LIN {X 0,Y 361.859,Z 339.019,A -85,B 0,C 180,E1 -13169.074,E2 -13169.074} C_VEL
LIN {X 0,Y 361.85,Z 339.033,A -85,B 0,C 180,E1 -13172.945,E2 -13172.945} C_VEL
LIN {X 0,Y 361.866,Z 339.018,A -85,B 0,C 180,E1 -13175.637,E2 -13175.637} C_VEL
LIN {X 0,Y 361.827,Z 339.039,A -85,B 0,C 180,E1 -13179.018,E2 -13179.018} C_VEL
LIN {X 0,Y 361.832,Z 339.037,A -85,B 0,C 180,E1 -13182.83,E2 -13182.83} C_VEL
LIN {X 0,Y 361.815,Z 339.032,A -85,B 0,C 180,E1 -13185.948,E2 -13185.948} C_VEL
LIN {X 0,Y 361.813,Z 339.037,A -85,B 0,C 180,E1 -13189.25,E2 -13189.25} C_VEL
LIN {X 0,Y 361.863,Z 339.037,A -85,B 0,C 180,E1 -13192.981,E2 -13192.981} C_VEL
LIN {X 0,Y 361.888,Z 339.154,A -85,B 0,C 180,E1 -13194.653,E2 -13194.653} C_VEL
LIN {X 0,Y 364.151,Z 348.355,A -85,B 0,C 180,E1 -13197.305,E2 -13197.305} C_VEL
LIN {X 0,Y 374.278,Z 371.025,A -85,B 0,C 180,E1 -13198.692,E2 -13198.692} C_VEL
LIN {X 0,Y 376.076,Z 376.225,A -85,B 0,C 180,E1 -13198.951,E2 -13198.951} C_VEL
LIN {X 0,Y 376.861,Z 380.502,A -85,B 0,C 180,E1 -13199.105,E2 -13199.105} C_VEL
LIN {X 0,Y 374.503,Z 484.658,A -85,B 0,C 180,E1 -13201.142,E2 -13201.142} C_VEL
LIN {X 0,Y 373.689,Z 499.489,A -85,B 0,C 180,E1 -13201.648,E2 -13201.648} C_VEL
LIN {X 0,Y 372.585,Z 513.31,A -85,B 0,C 180,E1 -13202.343,E2 -13202.343} C_VEL
LIN {X 0,Y 371.503,Z 525.302,A -85,B 0,C 180,E1 -13203.149,E2 -13203.149} C_VEL
LIN {X 0,Y 370.031,Z 538.195,A -85,B 0,C 180,E1 -13204.249,E2 -13204.249} C_VEL
LIN {X 0,Y 368.437,Z 549.874,A -85,B 0,C 180,E1 -13205.488,E2 -13205.488} C_VEL
LIN {X 0,Y 367.047,Z 560.816,A -85,B 0,C 180,E1 -13206.927,E2 -13206.927} C_VEL
LIN {X 0,Y 365.472,Z 571.118,A -85,B 0,C 180,E1 -13208.57,E2 -13208.57} C_VEL
LIN {X 0,Y 364.126,Z 579.801,A -85,B 0,C 180,E1 -13210.259,E2 -13210.259} C_VEL
LIN {X 0,Y 362.938,Z 588.089,A -85,B 0,C 180,E1 -13212.243,E2 -13212.243} C_VEL
LIN {X 0,Y 361.932,Z 594.713,A -85,B 0,C 180,E1 -13214.225,E2 -13214.225} C_VEL
LIN {X 0,Y 361.377,Z 599.273,A -85,B 0,C 180,E1 -13215.93,E2 -13215.93} C_VEL
LIN {X 0,Y 360.876,Z 602.89,A -85,B 0,C 180,E1 -13217.63,E2 -13217.63} C_VEL
LIN {X 0,Y 360.463,Z 606.411,A -85,B 0,C 180,E1 -13219.894,E2 -13219.894} C_VEL
LIN {X 0,Y 360.324,Z 608.525,A -85,B 0,C 180,E1 -13222.153,E2 -13222.153} C_VEL
LIN {X 0,Y 360.339,Z 609.296,A -85,B 0,C 180,E1 -13224.404,E2 -13224.404} C_VEL
LIN {X 0,Y 360.306,Z 608.752,A -85,B 0,C 180,E1 -13226.645,E2 -13226.645} C_VEL
LIN {X 0,Y 360.396,Z 606.887,A -85,B 0,C 180,E1 -13228.883,E2 -13228.883} C_VEL
LIN {X 0,Y 360.58,Z 603.647,A -85,B 0,C 180,E1 -13231.117,E2 -13231.117} C_VEL
LIN {X 0,Y 360.995,Z 598.934,A -85,B 0,C 180,E1 -13233.348,E2 -13233.348} C_VEL
LIN {X 0,Y 361.574,Z 594.379,A -85,B 0,C 180,E1 -13235.018,E2 -13235.018} C_VEL
LIN {X 0,Y 362.267,Z 587.776,A -85,B 0,C 180,E1 -13236.964,E2 -13236.964} C_VEL
LIN {X 0,Y 363.207,Z 579.566,A -85,B 0,C 180,E1 -13238.905,E2 -13238.905} C_VEL
LIN {X 0,Y 363.908,Z 572.559,A -85,B 0,C 180,E1 -13240.291,E2 -13240.291} C_VEL
LIN {X 0,Y 365.328,Z 562.556,A -85,B 0,C 180,E1 -13241.935,E2 -13241.935} C_VEL
LIN {X 0,Y 366.604,Z 551.394,A -85,B 0,C 180,E1 -13243.441,E2 -13243.441} C_VEL
LIN {X 0,Y 367.903,Z 538.895,A -85,B 0,C 180,E1 -13244.803,E2 -13244.803} C_VEL
LIN {X 0,Y 369.111,Z 526.476,A -85,B 0,C 180,E1 -13245.885,E2 -13245.885} C_VEL
LIN {X 0,Y 369.72,Z 519.402,A -85,B 0,C 180,E1 -13246.397,E2 -13246.397} C_VEL
LIN {X 0,Y 369.535,Z 514.034,A -85,B 0,C 180,E1 -13246.781,E2 -13246.781} C_VEL
LIN {X 0,Y 367.497,Z 505.26,A -85,B 0,C 180,E1 -13247.428,E2 -13247.428} C_VEL
LIN {X 0,Y 365.305,Z 496.282,A -85,B 0,C 180,E1 -13247.988,E2 -13247.988} C_VEL
LIN {X 0,Y 364.865,Z 490.597,A -85,B 0,C 180,E1 -13248.231,E2 -13248.231} C_VEL
LIN {X 0,Y 365.345,Z 475.344,A -85,B 0,C 180,E1 -13248.615,E2 -13248.615} C_VEL
LIN {X 0,Y 367.351,Z 379.982,A -85,B 0,C 180,E1 -13250.471,E2 -13250.471} C_VEL
LIN {X 0,Y 365.287,Z 370.104,A -85,B 0,C 180,E1 -13250.822,E2 -13250.822} C_VEL
LIN {X 0,Y 356.698,Z 348.251,A -85,B 0,C 180,E1 -13251.941,E2 -13251.941} C_VEL
LIN {X 0,Y 354.827,Z 339.915,A -85,B 0,C 180,E1 -13254.262,E2 -13254.262} C_VEL
LIN {X 0,Y 354.796,Z 339.921,A -85,B 0,C 180,E1 -13257.104,E2 -13257.104} C_VEL
LIN {X 0,Y 354.796,Z 339.911,A -85,B 0,C 180,E1 -13259.684,E2 -13259.684} C_VEL
LIN {X 0,Y 354.81,Z 339.912,A -85,B 0,C 180,E1 -13263.702,E2 -13263.702} C_VEL
LIN {X 0,Y 354.794,Z 339.916,A -85,B 0,C 180,E1 -13266.46,E2 -13266.46} C_VEL
LIN {X 0,Y 354.771,Z 339.916,A -85,B 0,C 180,E1 -13269.412,E2 -13269.412} C_VEL
LIN {X 0,Y 354.784,Z 339.918,A -85,B 0,C 180,E1 -13272.866,E2 -13272.866} C_VEL
LIN {X 0,Y 354.765,Z 339.916,A -85,B 0,C 180,E1 -13276.103,E2 -13276.103} C_VEL
LIN {X 0,Y 354.765,Z 339.916,A -85,B 0,C 180,E1 -13279.175,E2 -13279.175} C_VEL
LIN {X 0,Y 354.801,Z 339.91,A -85,B 0,C 180,E1 -13282.404,E2 -13282.404} C_VEL
LIN {X 0,Y 354.813,Z 339.913,A -85,B 0,C 180,E1 -13284.94,E2 -13284.94} C_VEL
LIN {X 0,Y 354.796,Z 339.91,A -85,B 0,C 180,E1 -13288.405,E2 -13288.405} C_VEL
LIN {X 0,Y 354.791,Z 339.91,A -85,B 0,C 180,E1 -13291.613,E2 -13291.613} C_VEL
LIN {X 0,Y 354.807,Z 339.912,A -85,B 0,C 180,E1 -13295.419,E2 -13295.419} C_VEL
LIN {X 0,Y 354.824,Z 339.888,A -85,B 0,C 180,E1 -13299.113,E2 -13299.113} C_VEL
LIN {X 0,Y 354.854,Z 339.907,A -85,B 0,C 180,E1 -13302.717,E2 -13302.717} C_VEL
LIN {X 0,Y 354.943,Z 339.89,A -85,B 0,C 180,E1 -13306.254,E2 -13306.254} C_VEL
LIN {X 0,Y 354.959,Z 339.867,A -85,B 0,C 180,E1 -13309.735,E2 -13309.735} C_VEL
LIN {X 0,Y 355.091,Z 339.875,A -85,B 0,C 180,E1 -13313.18,E2 -13313.18} C_VEL
LIN {X 0,Y 355.237,Z 339.857,A -85,B 0,C 180,E1 -13317.732,E2 -13317.732} C_VEL
LIN {X 0,Y 355.175,Z 339.859,A -85,B 0,C 180,E1 -13321.133,E2 -13321.133} C_VEL
LIN {X 0,Y 355.231,Z 339.861,A -85,B 0,C 180,E1 -13322.267,E2 -13322.267} C_VEL
LIN {X 0,Y 355.092,Z 339.875,A -85,B 0,C 180,E1 -13326.82,E2 -13326.82} C_VEL
LIN {X 0,Y 354.959,Z 339.892,A -85,B 0,C 180,E1 -13330.264,E2 -13330.264} C_VEL
LIN {X 0,Y 354.945,Z 339.893,A -85,B 0,C 180,E1 -13334.019,E2 -13334.019} C_VEL
LIN {X 0,Y 354.925,Z 339.896,A -85,B 0,C 180,E1 -13338.108,E2 -13338.108} C_VEL
LIN {X 0,Y 354.835,Z 339.908,A -85,B 0,C 180,E1 -13342.106,E2 -13342.106} C_VEL
LIN {X 0,Y 354.872,Z 339.905,A -85,B 0,C 180,E1 -13345.829,E2 -13345.829} C_VEL
LIN {X 0,Y 354.809,Z 339.913,A -85,B 0,C 180,E1 -13349.682,E2 -13349.682} C_VEL
LIN {X 0,Y 354.832,Z 339.914,A -85,B 0,C 180,E1 -13353.682,E2 -13353.682} C_VEL
LIN {X 0,Y 354.803,Z 339.915,A -85,B 0,C 180,E1 -13356.459,E2 -13356.459} C_VEL
LIN {X 0,Y 354.825,Z 339.913,A -85,B 0,C 180,E1 -13359.423,E2 -13359.423} C_VEL
LIN {X 0,Y 354.789,Z 339.917,A -85,B 0,C 180,E1 -13362.867,E2 -13362.867} C_VEL
LIN {X 0,Y 354.768,Z 339.918,A -85,B 0,C 180,E1 -13366.103,E2 -13366.103} C_VEL
LIN {X 0,Y 354.789,Z 339.918,A -85,B 0,C 180,E1 -13369.179,E2 -13369.179} C_VEL
LIN {X 0,Y 354.809,Z 339.918,A -85,B 0,C 180,E1 -13372.402,E2 -13372.402} C_VEL
LIN {X 0,Y 354.813,Z 339.918,A -85,B 0,C 180,E1 -13374.941,E2 -13374.941} C_VEL
LIN {X 0,Y 354.832,Z 339.964,A -85,B 0,C 180,E1 -13377.039,E2 -13377.039} C_VEL
LIN {X 0,Y 357.952,Z 353.28,A -85,B 0,C 180,E1 -13380.365,E2 -13380.365} C_VEL
LIN {X 0,Y 360.186,Z 364.464,A -85,B 0,C 180,E1 -13383.021,E2 -13383.021} C_VEL
LIN {X 0,Y 360.211,Z 366.003,A -85,B 0,C 180,E1 -13383.361,E2 -13383.361} C_VEL
LIN {X 0,Y 365.124,Z 394.057,A -85,B 0,C 180,E1 -13384.311,E2 -13384.311} C_VEL
LIN {X 0,Y 366.939,Z 405.452,A -85,B 0,C 180,E1 -13384.672,E2 -13384.672} C_VEL
LIN {X 0,Y 364.837,Z 504.382,A -85,B 0,C 180,E1 -13386.628,E2 -13386.628} C_VEL
LIN {X 0,Y 364.064,Z 518.99,A -85,B 0,C 180,E1 -13387.139,E2 -13387.139} C_VEL
LIN {X 0,Y 363.033,Z 532.395,A -85,B 0,C 180,E1 -13387.821,E2 -13387.821} C_VEL
LIN {X 0,Y 361.759,Z 546.228,A -85,B 0,C 180,E1 -13388.772,E2 -13388.772} C_VEL
LIN {X 0,Y 360.495,Z 558.957,A -85,B 0,C 180,E1 -13389.903,E2 -13389.903} C_VEL
LIN {X 0,Y 359.032,Z 570.399,A -85,B 0,C 180,E1 -13391.156,E2 -13391.156} C_VEL
LIN {X 0,Y 357.718,Z 580.918,A -85,B 0,C 180,E1 -13392.566,E2 -13392.566} C_VEL
LIN {X 0,Y 356.386,Z 591.377,A -85,B 0,C 180,E1 -13394.267,E2 -13394.267} C_VEL
LIN {X 0,Y 355.49,Z 600.131,A -85,B 0,C 180,E1 -13396.011,E2 -13396.011} C_VEL
LIN {X 0,Y 354.542,Z 608.246,A -85,B 0,C 180,E1 -13397.987,E2 -13397.987} C_VEL
LIN {X 0,Y 353.928,Z 614.029,A -85,B 0,C 180,E1 -13399.705,E2 -13399.705} C_VEL
LIN {X 0,Y 353.584,Z 618.743,A -85,B 0,C 180,E1 -13401.427,E2 -13401.427} C_VEL
LIN {X 0,Y 353.4,Z 622.55,A -85,B 0,C 180,E1 -13403.147,E2 -13403.147} C_VEL
LIN {X 0,Y 353.269,Z 626.266,A -85,B 0,C 180,E1 -13405.436,E2 -13405.436} C_VEL
LIN {X 0,Y 353.181,Z 628.562,A -85,B 0,C 180,E1 -13407.719,E2 -13407.719} C_VEL
LIN {X 0,Y 353.261,Z 629.505,A -85,B 0,C 180,E1 -13410,E2 -13410} C_VEL
LIN {X 0,Y 353.168,Z 629.106,A -85,B 0,C 180,E1 -13412.281,E2 -13412.281} C_VEL
LIN {X 0,Y 353.247,Z 627.377,A -85,B 0,C 180,E1 -13414.565,E2 -13414.565} C_VEL
LIN {X 0,Y 353.402,Z 624.276,A -85,B 0,C 180,E1 -13416.853,E2 -13416.853} C_VEL
LIN {X 0,Y 353.737,Z 619.722,A -85,B 0,C 180,E1 -13419.146,E2 -13419.146} C_VEL
LIN {X 0,Y 354.188,Z 615.221,A -85,B 0,C 180,E1 -13420.866,E2 -13420.866} C_VEL
LIN {X 0,Y 355.165,Z 608.756,A -85,B 0,C 180,E1 -13422.863,E2 -13422.863} C_VEL
LIN {X 0,Y 356.139,Z 600.743,A -85,B 0,C 180,E1 -13424.865,E2 -13424.865} C_VEL
LIN {X 0,Y 357.459,Z 592.378,A -85,B 0,C 180,E1 -13426.564,E2 -13426.564} C_VEL
LIN {X 0,Y 359.051,Z 582.325,A -85,B 0,C 180,E1 -13428.251,E2 -13428.251} C_VEL
LIN {X 0,Y 360.848,Z 571.117,A -85,B 0,C 180,E1 -13429.78,E2 -13429.78} C_VEL
LIN {X 0,Y 362.413,Z 559.991,A -85,B 0,C 180,E1 -13431.024,E2 -13431.024} C_VEL
LIN {X 0,Y 363.899,Z 547.901,A -85,B 0,C 180,E1 -13432.123,E2 -13432.123} C_VEL
LIN {X 0,Y 365.294,Z 534.497,A -85,B 0,C 180,E1 -13433.079,E2 -13433.079} C_VEL
LIN {X 0,Y 366.594,Z 520.522,A -85,B 0,C 180,E1 -13433.816,E2 -13433.816} C_VEL
LIN {X 0,Y 367.603,Z 505.812,A -85,B 0,C 180,E1 -13434.346,E2 -13434.346} C_VEL
LIN {X 0,Y 368.3,Z 480.796,A -85,B 0,C 180,E1 -13434.88,E2 -13434.88} C_VEL
LIN {X 0,Y 370.024,Z 405.562,A -85,B 0,C 180,E1 -13436.358,E2 -13436.358} C_VEL
LIN {X 0,Y 365.249,Z 380.502,A -85,B 0,C 180,E1 -13437.31,E2 -13437.31} C_VEL
LIN {X 0,Y 362.8,Z 370.211,A -85,B 0,C 180,E1 -13437.754,E2 -13437.754} C_VEL
LIN {X 0,Y 361.042,Z 365.698,A -85,B 0,C 180,E1 -13438.034,E2 -13438.034} C_VEL
LIN {X 0,Y 358.46,Z 354.094,A -85,B 0,C 180,E1 -13440.975,E2 -13440.975} C_VEL
LIN {X 0,Y 355.248,Z 341.576,A -85,B 0,C 180,E1 -13444.352,E2 -13444.352} C_VEL
LIN {X 0,Y 354.84,Z 339.909,A -85,B 0,C 180,E1 -13444.85,E2 -13444.85} C_VEL
LIN {X 0,Y 354.806,Z 339.908,A -85,B 0,C 180,E1 -13447.883,E2 -13447.883} C_VEL
LIN {X 0,Y 354.789,Z 339.914,A -85,B 0,C 180,E1 -13451.172,E2 -13451.172} C_VEL
LIN {X 0,Y 354.765,Z 339.921,A -85,B 0,C 180,E1 -13454.507,E2 -13454.507} C_VEL
LIN {X 0,Y 354.796,Z 339.913,A -85,B 0,C 180,E1 -13457.663,E2 -13457.663} C_VEL
LIN {X 0,Y 354.817,Z 339.908,A -85,B 0,C 180,E1 -13460.666,E2 -13460.666} C_VEL
LIN {X 0,Y 354.824,Z 339.909,A -85,B 0,C 180,E1 -13464.301,E2 -13464.301} C_VEL
LIN {X 0,Y 354.789,Z 339.912,A -85,B 0,C 180,E1 -13467.667,E2 -13467.667} C_VEL
LIN {X 0,Y 354.805,Z 339.912,A -85,B 0,C 180,E1 -13471.615,E2 -13471.615} C_VEL
LIN {X 0,Y 354.854,Z 339.906,A -85,B 0,C 180,E1 -13475.423,E2 -13475.423} C_VEL
LIN {X 0,Y 354.829,Z 339.908,A -85,B 0,C 180,E1 -13479.114,E2 -13479.114} C_VEL
LIN {X 0,Y 354.902,Z 339.896,A -85,B 0,C 180,E1 -13482.72,E2 -13482.72} C_VEL
LIN {X 0,Y 354.954,Z 339.887,A -85,B 0,C 180,E1 -13486.256,E2 -13486.256} C_VEL
LIN {X 0,Y 354.979,Z 339.894,A -85,B 0,C 180,E1 -13489.736,E2 -13489.736} C_VEL
LIN {X 0,Y 355.092,Z 339.874,A -85,B 0,C 180,E1 -13493.18,E2 -13493.18} C_VEL
LIN {X 0,Y 355.231,Z 339.854,A -85,B 0,C 180,E1 -13497.733,E2 -13497.733} C_VEL
LIN {X 0,Y 355.149,Z 339.865,A -85,B 0,C 180,E1 -13501.134,E2 -13501.134} C_VEL
LIN {X 0,Y 355.237,Z 339.853,A -85,B 0,C 180,E1 -13502.268,E2 -13502.268} C_VEL
LIN {X 0,Y 355.091,Z 339.866,A -85,B 0,C 180,E1 -13506.82,E2 -13506.82} C_VEL
LIN {X 0,Y 354.959,Z 339.891,A -85,B 0,C 180,E1 -13510.265,E2 -13510.265} C_VEL
LIN {X 0,Y 354.927,Z 339.9,A -85,B 0,C 180,E1 -13514.006,E2 -13514.006} C_VEL
LIN {X 0,Y 354.845,Z 339.91,A -85,B 0,C 180,E1 -13518.068,E2 -13518.068} C_VEL
LIN {X 0,Y 354.809,Z 339.913,A -85,B 0,C 180,E1 -13522.108,E2 -13522.108} C_VEL
LIN {X 0,Y 354.802,Z 339.913,A -85,B 0,C 180,E1 -13525.835,E2 -13525.835} C_VEL
LIN {X 0,Y 354.796,Z 339.89,A -85,B 0,C 180,E1 -13529.684,E2 -13529.684} C_VEL
LIN {X 0,Y 354.81,Z 339.914,A -85,B 0,C 180,E1 -13533.702,E2 -13533.702} C_VEL
LIN {X 0,Y 354.794,Z 339.894,A -85,B 0,C 180,E1 -13536.46,E2 -13536.46} C_VEL
LIN {X 0,Y 354.771,Z 339.92,A -85,B 0,C 180,E1 -13539.413,E2 -13539.413} C_VEL
LIN {X 0,Y 354.784,Z 339.915,A -85,B 0,C 180,E1 -13542.866,E2 -13542.866} C_VEL
LIN {X 0,Y 354.765,Z 339.91,A -85,B 0,C 180,E1 -13546.103,E2 -13546.103} C_VEL
LIN {X 0,Y 354.765,Z 339.914,A -85,B 0,C 180,E1 -13549.175,E2 -13549.175} C_VEL
LIN {X 0,Y 354.801,Z 339.919,A -85,B 0,C 180,E1 -13552.405,E2 -13552.405} C_VEL
LIN {X 0,Y 354.82,Z 339.929,A -85,B 0,C 180,E1 -13554.078,E2 -13554.078} C_VEL
LIN {X 0,Y 357.07,Z 348.881,A -85,B 0,C 180,E1 -13556.675,E2 -13556.675} C_VEL
LIN {X 0,Y 367.365,Z 371.416,A -85,B 0,C 180,E1 -13558.113,E2 -13558.113} C_VEL
LIN {X 0,Y 370.031,Z 378.402,A -85,B 0,C 180,E1 -13558.494,E2 -13558.494} C_VEL
LIN {X 0,Y 370.558,Z 380.853,A -85,B 0,C 180,E1 -13558.592,E2 -13558.592} C_VEL
LIN {X 0,Y 368.133,Z 485.217,A -85,B 0,C 180,E1 -13560.672,E2 -13560.672} C_VEL
LIN {X 0,Y 367.285,Z 499.917,A -85,B 0,C 180,E1 -13561.186,E2 -13561.186} C_VEL
LIN {X 0,Y 366.076,Z 514.353,A -85,B 0,C 180,E1 -13561.932,E2 -13561.932} C_VEL
LIN {X 0,Y 364.921,Z 526.525,A -85,B 0,C 180,E1 -13562.78,E2 -13562.78} C_VEL
LIN {X 0,Y 363.368,Z 539.217,A -85,B 0,C 180,E1 -13563.895,E2 -13563.895} C_VEL
LIN {X 0,Y 361.729,Z 550.749,A -85,B 0,C 180,E1 -13565.156,E2 -13565.156} C_VEL
LIN {X 0,Y 360.277,Z 561.477,A -85,B 0,C 180,E1 -13566.605,E2 -13566.605} C_VEL
LIN {X 0,Y 358.759,Z 570.966,A -85,B 0,C 180,E1 -13568.148,E2 -13568.148} C_VEL
LIN {X 0,Y 357.333,Z 579.709,A -85,B 0,C 180,E1 -13569.868,E2 -13569.868} C_VEL
LIN {X 0,Y 356.045,Z 588.064,A -85,B 0,C 180,E1 -13571.887,E2 -13571.887} C_VEL
LIN {X 0,Y 355.007,Z 594.739,A -85,B 0,C 180,E1 -13573.909,E2 -13573.909} C_VEL
LIN {X 0,Y 354.203,Z 600.635,A -85,B 0,C 180,E1 -13576.225,E2 -13576.225} C_VEL
LIN {X 0,Y 353.61,Z 604.938,A -85,B 0,C 180,E1 -13578.536,E2 -13578.536} C_VEL
LIN {X 0,Y 353.304,Z 607.78,A -85,B 0,C 180,E1 -13580.843,E2 -13580.843} C_VEL
LIN {X 0,Y 353.272,Z 609.251,A -85,B 0,C 180,E1 -13583.145,E2 -13583.145} C_VEL
LIN {X 0,Y 353.246,Z 609.398,A -85,B 0,C 180,E1 -13585.435,E2 -13585.435} C_VEL
LIN {X 0,Y 353.231,Z 608.232,A -85,B 0,C 180,E1 -13587.719,E2 -13587.719} C_VEL
LIN {X 0,Y 353.377,Z 605.734,A -85,B 0,C 180,E1 -13590,E2 -13590} C_VEL
LIN {X 0,Y 353.66,Z 601.817,A -85,B 0,C 180,E1 -13592.278,E2 -13592.278} C_VEL
LIN {X 0,Y 354.257,Z 596.358,A -85,B 0,C 180,E1 -13594.551,E2 -13594.551} C_VEL
LIN {X 0,Y 354.939,Z 591.191,A -85,B 0,C 180,E1 -13596.252,E2 -13596.252} C_VEL
LIN {X 0,Y 355.731,Z 583.754,A -85,B 0,C 180,E1 -13598.235,E2 -13598.235} C_VEL
LIN {X 0,Y 356.581,Z 575.956,A -85,B 0,C 180,E1 -13599.944,E2 -13599.944} C_VEL
LIN {X 0,Y 357.907,Z 566.674,A -85,B 0,C 180,E1 -13601.611,E2 -13601.611} C_VEL
LIN {X 0,Y 359.266,Z 556.341,A -85,B 0,C 180,E1 -13603.145,E2 -13603.145} C_VEL
LIN {X 0,Y 360.581,Z 544.953,A -85,B 0,C 180,E1 -13604.533,E2 -13604.533} C_VEL
LIN {X 0,Y 361.742,Z 533.902,A -85,B 0,C 180,E1 -13605.639,E2 -13605.639} C_VEL
LIN {X 0,Y 362.846,Z 522.03,A -85,B 0,C 180,E1 -13606.6,E2 -13606.6} C_VEL
LIN {X 0,Y 363.89,Z 509.031,A -85,B 0,C 180,E1 -13607.419,E2 -13607.419} C_VEL
LIN {X 0,Y 364.694,Z 495.02,A -85,B 0,C 180,E1 -13608.068,E2 -13608.068} C_VEL
LIN {X 0,Y 364.865,Z 490.597,A -85,B 0,C 180,E1 -13608.231,E2 -13608.231} C_VEL
LIN {X 0,Y 364.409,Z 484.85,A -85,B 0,C 180,E1 -13608.447,E2 -13608.447} C_VEL
LIN {X 0,Y 359.505,Z 466.196,A -85,B 0,C 180,E1 -13609.185,E2 -13609.185} C_VEL
LIN {X 0,Y 359.112,Z 460.384,A -85,B 0,C 180,E1 -13609.331,E2 -13609.331} C_VEL
LIN {X 0,Y 360.741,Z 380.031,A -85,B 0,C 180,E1 -13610.932,E2 -13610.932} C_VEL
LIN {X 0,Y 359.001,Z 372.319,A -85,B 0,C 180,E1 -13611.222,E2 -13611.222} C_VEL
LIN {X 0,Y 350.657,Z 351.352,A -85,B 0,C 180,E1 -13612.308,E2 -13612.308} C_VEL
LIN {X 0,Y 349.52,Z 348.57,A -85,B 0,C 180,E1 -13612.46,E2 -13612.46} C_VEL
LIN {X 0,Y 347.76,Z 340.795,A -85,B 0,C 180,E1 -13614.699,E2 -13614.699} C_VEL
LIN {X 0,Y 347.727,Z 340.798,A -85,B 0,C 180,E1 -13617.701,E2 -13617.701} C_VEL
LIN {X 0,Y 347.732,Z 340.789,A -85,B 0,C 180,E1 -13620.35,E2 -13620.35} C_VEL
LIN {X 0,Y 347.751,Z 340.792,A -85,B 0,C 180,E1 -13624.043,E2 -13624.043} C_VEL
LIN {X 0,Y 347.757,Z 340.792,A -85,B 0,C 180,E1 -13627.322,E2 -13627.322} C_VEL
LIN {X 0,Y 347.699,Z 340.799,A -85,B 0,C 180,E1 -13630.302,E2 -13630.302} C_VEL
LIN {X 0,Y 347.723,Z 340.795,A -85,B 0,C 180,E1 -13633.408,E2 -13633.408} C_VEL
LIN {X 0,Y 347.725,Z 340.799,A -85,B 0,C 180,E1 -13636.687,E2 -13636.687} C_VEL
LIN {X 0,Y 347.703,Z 340.797,A -85,B 0,C 180,E1 -13640.182,E2 -13640.182} C_VEL
LIN {X 0,Y 347.758,Z 340.787,A -85,B 0,C 180,E1 -13642.678,E2 -13642.678} C_VEL
LIN {X 0,Y 347.751,Z 340.791,A -85,B 0,C 180,E1 -13645.956,E2 -13645.956} C_VEL
LIN {X 0,Y 347.738,Z 340.792,A -85,B 0,C 180,E1 -13649.651,E2 -13649.651} C_VEL
LIN {X 0,Y 347.737,Z 340.787,A -85,B 0,C 180,E1 -13653.6,E2 -13653.6} C_VEL
LIN {X 0,Y 347.754,Z 340.794,A -85,B 0,C 180,E1 -13656.159,E2 -13656.159} C_VEL
LIN {X 0,Y 347.774,Z 340.764,A -85,B 0,C 180,E1 -13659.907,E2 -13659.907} C_VEL
LIN {X 0,Y 347.8,Z 340.784,A -85,B 0,C 180,E1 -13663.566,E2 -13663.566} C_VEL
LIN {X 0,Y 347.89,Z 340.761,A -85,B 0,C 180,E1 -13667.16,E2 -13667.16} C_VEL
LIN {X 0,Y 347.938,Z 340.753,A -85,B 0,C 180,E1 -13670.7,E2 -13670.7} C_VEL
LIN {X 0,Y 348.044,Z 340.758,A -85,B 0,C 180,E1 -13674.205,E2 -13674.205} C_VEL
LIN {X 0,Y 348.198,Z 340.734,A -85,B 0,C 180,E1 -13677.686,E2 -13677.686} C_VEL
LIN {X 0,Y 348.144,Z 340.735,A -85,B 0,C 180,E1 -13681.156,E2 -13681.156} C_VEL
LIN {X 0,Y 348.192,Z 340.739,A -85,B 0,C 180,E1 -13682.313,E2 -13682.313} C_VEL
LIN {X 0,Y 348.058,Z 340.751,A -85,B 0,C 180,E1 -13686.958,E2 -13686.958} C_VEL
LIN {X 0,Y 347.899,Z 340.771,A -85,B 0,C 180,E1 -13690.475,E2 -13690.475} C_VEL
LIN {X 0,Y 347.901,Z 340.77,A -85,B 0,C 180,E1 -13694.149,E2 -13694.149} C_VEL
LIN {X 0,Y 347.893,Z 340.771,A -85,B 0,C 180,E1 -13698.29,E2 -13698.29} C_VEL
LIN {X 0,Y 347.79,Z 340.787,A -85,B 0,C 180,E1 -13701.634,E2 -13701.634} C_VEL
LIN {X 0,Y 347.798,Z 340.785,A -85,B 0,C 180,E1 -13705.109,E2 -13705.109} C_VEL
LIN {X 0,Y 347.784,Z 340.793,A -85,B 0,C 180,E1 -13707.696,E2 -13707.696} C_VEL
LIN {X 0,Y 347.746,Z 340.794,A -85,B 0,C 180,E1 -13710.348,E2 -13710.348} C_VEL
LIN {X 0,Y 347.75,Z 340.796,A -85,B 0,C 180,E1 -13714.043,E2 -13714.043} C_VEL
LIN {X 0,Y 347.767,Z 340.795,A -85,B 0,C 180,E1 -13717.32,E2 -13717.32} C_VEL
LIN {X 0,Y 347.734,Z 340.795,A -85,B 0,C 180,E1 -13720.297,E2 -13720.297} C_VEL
LIN {X 0,Y 347.724,Z 340.799,A -85,B 0,C 180,E1 -13723.408,E2 -13723.408} C_VEL
LIN {X 0,Y 347.726,Z 340.795,A -85,B 0,C 180,E1 -13726.686,E2 -13726.686} C_VEL
LIN {X 0,Y 347.748,Z 340.795,A -85,B 0,C 180,E1 -13730.173,E2 -13730.173} C_VEL
LIN {X 0,Y 347.763,Z 340.796,A -85,B 0,C 180,E1 -13732.679,E2 -13732.679} C_VEL
LIN {X 0,Y 347.796,Z 340.793,A -85,B 0,C 180,E1 -13736.446,E2 -13736.446} C_VEL
LIN {X 0,Y 347.789,Z 340.875,A -85,B 0,C 180,E1 -13736.608,E2 -13736.608} C_VEL
LIN {X 0,Y 350.861,Z 353.898,A -85,B 0,C 180,E1 -13739.949,E2 -13739.949} C_VEL
LIN {X 0,Y 353.272,Z 365.799,A -85,B 0,C 180,E1 -13742.843,E2 -13742.843} C_VEL
LIN {X 0,Y 355.599,Z 377.105,A -85,B 0,C 180,E1 -13743.272,E2 -13743.272} C_VEL
LIN {X 0,Y 360.4,Z 405.777,A -85,B 0,C 180,E1 -13744.233,E2 -13744.233} C_VEL
LIN {X 0,Y 358.255,Z 504.083,A -85,B 0,C 180,E1 -13746.21,E2 -13746.21} C_VEL
LIN {X 0,Y 357.521,Z 517.96,A -85,B 0,C 180,E1 -13746.696,E2 -13746.696} C_VEL
LIN {X 0,Y 356.441,Z 531.579,A -85,B 0,C 180,E1 -13747.388,E2 -13747.388} C_VEL
LIN {X 0,Y 355.208,Z 544.43,A -85,B 0,C 180,E1 -13748.265,E2 -13748.265} C_VEL
LIN {X 0,Y 353.945,Z 556.93,A -85,B 0,C 180,E1 -13749.363,E2 -13749.363} C_VEL
LIN {X 0,Y 352.462,Z 568.698,A -85,B 0,C 180,E1 -13750.64,E2 -13750.64} C_VEL
LIN {X 0,Y 351.141,Z 578.482,A -85,B 0,C 180,E1 -13751.927,E2 -13751.927} C_VEL
LIN {X 0,Y 349.727,Z 589.315,A -85,B 0,C 180,E1 -13753.66,E2 -13753.66} C_VEL
LIN {X 0,Y 348.69,Z 597.964,A -85,B 0,C 180,E1 -13755.343,E2 -13755.343} C_VEL
LIN {X 0,Y 347.794,Z 605.69,A -85,B 0,C 180,E1 -13757.157,E2 -13757.157} C_VEL
LIN {X 0,Y 347.077,Z 611.877,A -85,B 0,C 180,E1 -13758.909,E2 -13758.909} C_VEL
LIN {X 0,Y 346.515,Z 618.446,A -85,B 0,C 180,E1 -13761.25,E2 -13761.25} C_VEL
LIN {X 0,Y 346.324,Z 622.277,A -85,B 0,C 180,E1 -13763.006,E2 -13763.006} C_VEL
LIN {X 0,Y 346.168,Z 626.016,A -85,B 0,C 180,E1 -13765.342,E2 -13765.342} C_VEL
LIN {X 0,Y 346.091,Z 628.335,A -85,B 0,C 180,E1 -13767.672,E2 -13767.672} C_VEL
LIN {X 0,Y 346.163,Z 629.298,A -85,B 0,C 180,E1 -13770,E2 -13770} C_VEL
LIN {X 0,Y 346.08,Z 628.921,A -85,B 0,C 180,E1 -13772.328,E2 -13772.328} C_VEL
LIN {X 0,Y 346.146,Z 627.211,A -85,B 0,C 180,E1 -13774.658,E2 -13774.658} C_VEL
LIN {X 0,Y 346.326,Z 624.133,A -85,B 0,C 180,E1 -13776.994,E2 -13776.994} C_VEL
LIN {X 0,Y 346.694,Z 619.604,A -85,B 0,C 180,E1 -13779.333,E2 -13779.333} C_VEL
LIN {X 0,Y 347.17,Z 615.126,A -85,B 0,C 180,E1 -13781.088,E2 -13781.088} C_VEL
LIN {X 0,Y 348.213,Z 608.688,A -85,B 0,C 180,E1 -13783.124,E2 -13783.124} C_VEL
LIN {X 0,Y 349.245,Z 600.706,A -85,B 0,C 180,E1 -13785.165,E2 -13785.165} C_VEL
LIN {X 0,Y 350.616,Z 592.375,A -85,B 0,C 180,E1 -13786.897,E2 -13786.897} C_VEL
LIN {X 0,Y 352.295,Z 582.364,A -85,B 0,C 180,E1 -13788.614,E2 -13788.614} C_VEL
LIN {X 0,Y 353.967,Z 572.308,A -85,B 0,C 180,E1 -13790.029,E2 -13790.029} C_VEL
LIN {X 0,Y 355.776,Z 560.313,A -85,B 0,C 180,E1 -13791.419,E2 -13791.419} C_VEL
LIN {X 0,Y 357.345,Z 548.175,A -85,B 0,C 180,E1 -13792.551,E2 -13792.551} C_VEL
LIN {X 0,Y 358.798,Z 534.91,A -85,B 0,C 180,E1 -13793.522,E2 -13793.522} C_VEL
LIN {X 0,Y 360.155,Z 521.147,A -85,B 0,C 180,E1 -13794.269,E2 -13794.269} C_VEL
LIN {X 0,Y 361.169,Z 506.851,A -85,B 0,C 180,E1 -13794.809,E2 -13794.809} C_VEL
LIN {X 0,Y 361.829,Z 487.006,A -85,B 0,C 180,E1 -13795.259,E2 -13795.259} C_VEL
LIN {X 0,Y 363.78,Z 406.899,A -85,B 0,C 180,E1 -13796.855,E2 -13796.855} C_VEL
LIN {X 0,Y 359.235,Z 382.593,A -85,B 0,C 180,E1 -13797.798,E2 -13797.798} C_VEL
LIN {X 0,Y 356.948,Z 372.933,A -85,B 0,C 180,E1 -13798.226,E2 -13798.226} C_VEL
LIN {X 0,Y 353.833,Z 365.502,A -85,B 0,C 180,E1 -13798.702,E2 -13798.702} C_VEL
LIN {X 0,Y 350.914,Z 352.92,A -85,B 0,C 180,E1 -13802.007,E2 -13802.007} C_VEL
LIN {X 0,Y 348.372,Z 343.099,A -85,B 0,C 180,E1 -13804.744,E2 -13804.744} C_VEL
LIN {X 0,Y 347.777,Z 340.791,A -85,B 0,C 180,E1 -13805.432,E2 -13805.432} C_VEL
LIN {X 0,Y 347.753,Z 340.782,A -85,B 0,C 180,E1 -13808.793,E2 -13808.793} C_VEL
LIN {X 0,Y 347.752,Z 340.791,A -85,B 0,C 180,E1 -13811.831,E2 -13811.831} C_VEL
LIN {X 0,Y 347.707,Z 340.796,A -85,B 0,C 180,E1 -13815.027,E2 -13815.027} C_VEL
LIN {X 0,Y 347.752,Z 340.789,A -85,B 0,C 180,E1 -13818.397,E2 -13818.397} C_VEL
LIN {X 0,Y 347.778,Z 340.788,A -85,B 0,C 180,E1 -13822.011,E2 -13822.011} C_VEL
LIN {X 0,Y 347.746,Z 340.792,A -85,B 0,C 180,E1 -13825.537,E2 -13825.537} C_VEL
LIN {X 0,Y 347.747,Z 340.795,A -85,B 0,C 180,E1 -13828.301,E2 -13828.301} C_VEL
LIN {X 0,Y 347.749,Z 340.791,A -85,B 0,C 180,E1 -13830.985,E2 -13830.985} C_VEL
LIN {X 0,Y 347.761,Z 340.786,A -85,B 0,C 180,E1 -13833.602,E2 -13833.602} C_VEL
LIN {X 0,Y 347.776,Z 340.791,A -85,B 0,C 180,E1 -13836.161,E2 -13836.161} C_VEL
LIN {X 0,Y 347.814,Z 340.785,A -85,B 0,C 180,E1 -13839.91,E2 -13839.91} C_VEL
LIN {X 0,Y 347.869,Z 340.77,A -85,B 0,C 180,E1 -13842.36,E2 -13842.36} C_VEL
LIN {X 0,Y 347.9,Z 340.768,A -85,B 0,C 180,E1 -13845.971,E2 -13845.971} C_VEL
LIN {X 0,Y 347.93,Z 340.77,A -85,B 0,C 180,E1 -13849.526,E2 -13849.526} C_VEL
LIN {X 0,Y 348.059,Z 340.75,A -85,B 0,C 180,E1 -13853.042,E2 -13853.042} C_VEL
LIN {X 0,Y 348.192,Z 340.73,A -85,B 0,C 180,E1 -13857.687,E2 -13857.687} C_VEL
LIN {X 0,Y 348.121,Z 340.74,A -85,B 0,C 180,E1 -13861.157,E2 -13861.157} C_VEL
LIN {X 0,Y 348.199,Z 340.729,A -85,B 0,C 180,E1 -13862.314,E2 -13862.314} C_VEL
LIN {X 0,Y 348.058,Z 340.742,A -85,B 0,C 180,E1 -13866.959,E2 -13866.959} C_VEL
LIN {X 0,Y 347.9,Z 340.769,A -85,B 0,C 180,E1 -13870.476,E2 -13870.476} C_VEL
LIN {X 0,Y 347.883,Z 340.776,A -85,B 0,C 180,E1 -13874.137,E2 -13874.137} C_VEL
LIN {X 0,Y 347.796,Z 340.787,A -85,B 0,C 180,E1 -13878.241,E2 -13878.241} C_VEL
LIN {X 0,Y 347.766,Z 340.786,A -85,B 0,C 180,E1 -13881.624,E2 -13881.624} C_VEL
LIN {X 0,Y 347.74,Z 340.787,A -85,B 0,C 180,E1 -13885.115,E2 -13885.115} C_VEL
LIN {X 0,Y 347.728,Z 340.792,A -85,B 0,C 180,E1 -13887.702,E2 -13887.702} C_VEL
LIN {X 0,Y 347.732,Z 340.767,A -85,B 0,C 180,E1 -13890.35,E2 -13890.35} C_VEL
LIN {X 0,Y 347.751,Z 340.791,A -85,B 0,C 180,E1 -13894.044,E2 -13894.044} C_VEL
LIN {X 0,Y 347.757,Z 340.774,A -85,B 0,C 180,E1 -13897.322,E2 -13897.322} C_VEL
LIN {X 0,Y 347.699,Z 340.795,A -85,B 0,C 180,E1 -13900.302,E2 -13900.302} C_VEL
LIN {X 0,Y 347.724,Z 340.798,A -85,B 0,C 180,E1 -13903.409,E2 -13903.409} C_VEL
LIN {X 0,Y 347.725,Z 340.791,A -85,B 0,C 180,E1 -13906.687,E2 -13906.687} C_VEL
LIN {X 0,Y 347.704,Z 340.798,A -85,B 0,C 180,E1 -13910.183,E2 -13910.183} C_VEL
LIN {X 0,Y 347.783,Z 340.891,A -85,B 0,C 180,E1 -13913.533,E2 -13913.533} C_VEL
LIN {X 0,Y 349.811,Z 348.899,A -85,B 0,C 180,E1 -13915.97,E2 -13915.97} C_VEL
LIN {X 0,Y 359.584,Z 369.858,A -85,B 0,C 180,E1 -13917.386,E2 -13917.386} C_VEL
LIN {X 0,Y 364.06,Z 380.926,A -85,B 0,C 180,E1 -13918.034,E2 -13918.034} C_VEL
LIN {X 0,Y 364.3,Z 384.253,A -85,B 0,C 180,E1 -13918.129,E2 -13918.129} C_VEL
LIN {X 0,Y 361.796,Z 484.505,A -85,B 0,C 180,E1 -13920.147,E2 -13920.147} C_VEL
LIN {X 0,Y 361.029,Z 498.814,A -85,B 0,C 180,E1 -13920.638,E2 -13920.638} C_VEL
LIN {X 0,Y 359.892,Z 512.257,A -85,B 0,C 180,E1 -13921.313,E2 -13921.313} C_VEL
LIN {X 0,Y 358.701,Z 524.178,A -85,B 0,C 180,E1 -13922.109,E2 -13922.109} C_VEL
LIN {X 0,Y 357.13,Z 537.368,A -85,B 0,C 180,E1 -13923.246,E2 -13923.246} C_VEL
LIN {X 0,Y 355.439,Z 549.267,A -85,B 0,C 180,E1 -13924.529,E2 -13924.529} C_VEL
LIN {X 0,Y 353.925,Z 559.427,A -85,B 0,C 180,E1 -13925.869,E2 -13925.869} C_VEL
LIN {X 0,Y 352.385,Z 569.181,A -85,B 0,C 180,E1 -13927.423,E2 -13927.423} C_VEL
LIN {X 0,Y 350.8,Z 578.257,A -85,B 0,C 180,E1 -13929.169,E2 -13929.169} C_VEL
LIN {X 0,Y 349.342,Z 586.911,A -85,B 0,C 180,E1 -13931.223,E2 -13931.223} C_VEL
LIN {X 0,Y 348.368,Z 592.959,A -85,B 0,C 180,E1 -13932.991,E2 -13932.991} C_VEL
LIN {X 0,Y 347.616,Z 597.945,A -85,B 0,C 180,E1 -13934.762,E2 -13934.762} C_VEL
LIN {X 0,Y 346.853,Z 603.064,A -85,B 0,C 180,E1 -13937.121,E2 -13937.121} C_VEL
LIN {X 0,Y 346.334,Z 606.66,A -85,B 0,C 180,E1 -13939.477,E2 -13939.477} C_VEL
LIN {X 0,Y 346.168,Z 608.843,A -85,B 0,C 180,E1 -13941.83,E2 -13941.83} C_VEL
LIN {X 0,Y 346.184,Z 609.681,A -85,B 0,C 180,E1 -13944.174,E2 -13944.174} C_VEL
LIN {X 0,Y 346.147,Z 609.206,A -85,B 0,C 180,E1 -13946.508,E2 -13946.508} C_VEL
LIN {X 0,Y 346.196,Z 607.415,A -85,B 0,C 180,E1 -13948.837,E2 -13948.837} C_VEL
LIN {X 0,Y 346.421,Z 604.267,A -85,B 0,C 180,E1 -13951.162,E2 -13951.162} C_VEL
LIN {X 0,Y 346.853,Z 599.643,A -85,B 0,C 180,E1 -13953.485,E2 -13953.485} C_VEL
LIN {X 0,Y 347.493,Z 595.128,A -85,B 0,C 180,E1 -13955.222,E2 -13955.222} C_VEL
LIN {X 0,Y 348.209,Z 588.619,A -85,B 0,C 180,E1 -13957.247,E2 -13957.247} C_VEL
LIN {X 0,Y 349.25,Z 580.545,A -85,B 0,C 180,E1 -13959.264,E2 -13959.264} C_VEL
LIN {X 0,Y 350.013,Z 573.597,A -85,B 0,C 180,E1 -13960.704,E2 -13960.704} C_VEL
LIN {X 0,Y 351.535,Z 563.72,A -85,B 0,C 180,E1 -13962.411,E2 -13962.411} C_VEL
LIN {X 0,Y 352.892,Z 552.763,A -85,B 0,C 180,E1 -13963.974,E2 -13963.974} C_VEL
LIN {X 0,Y 354.298,Z 540.509,A -85,B 0,C 180,E1 -13965.386,E2 -13965.386} C_VEL
LIN {X 0,Y 355.587,Z 528.376,A -85,B 0,C 180,E1 -13966.506,E2 -13966.506} C_VEL
LIN {X 0,Y 356.746,Z 514.911,A -85,B 0,C 180,E1 -13967.483,E2 -13967.483} C_VEL
LIN {X 0,Y 357.815,Z 500.747,A -85,B 0,C 180,E1 -13968.242,E2 -13968.242} C_VEL
LIN {X 0,Y 358.439,Z 486.791,A -85,B 0,C 180,E1 -13968.765,E2 -13968.765} C_VEL
LIN {X 0,Y 359.112,Z 460.384,A -85,B 0,C 180,E1 -13969.331,E2 -13969.331} C_VEL
LIN {X 0,Y 358.701,Z 454.573,A -85,B 0,C 180,E1 -13969.482,E2 -13969.482} C_VEL
LIN {X 0,Y 353.746,Z 435.901,A -85,B 0,C 180,E1 -13970.223,E2 -13970.223} C_VEL
LIN {X 0,Y 353.26,Z 430.089,A -85,B 0,C 180,E1 -13970.383,E2 -13970.383} C_VEL
LIN {X 0,Y 354.258,Z 381.129,A -85,B 0,C 180,E1 -13971.378,E2 -13971.378} C_VEL
LIN {X 0,Y 352.777,Z 374.676,A -85,B 0,C 180,E1 -13971.63,E2 -13971.63} C_VEL
LIN {X 0,Y 344.676,Z 354.391,A -85,B 0,C 180,E1 -13972.713,E2 -13972.713} C_VEL
LIN {X 0,Y 342.365,Z 348.702,A -85,B 0,C 180,E1 -13973.053,E2 -13973.053} C_VEL
LIN {X 0,Y 340.718,Z 341.673,A -85,B 0,C 180,E1 -13975.122,E2 -13975.122} C_VEL
LIN {X 0,Y 340.678,Z 341.676,A -85,B 0,C 180,E1 -13978.325,E2 -13978.325} C_VEL
LIN {X 0,Y 340.685,Z 341.671,A -85,B 0,C 180,E1 -13981.046,E2 -13981.046} C_VEL
LIN {X 0,Y 340.718,Z 341.669,A -85,B 0,C 180,E1 -13985.279,E2 -13985.279} C_VEL
LIN {X 0,Y 340.696,Z 341.673,A -85,B 0,C 180,E1 -13988.382,E2 -13988.382} C_VEL
LIN {X 0,Y 340.693,Z 341.668,A -85,B 0,C 180,E1 -13992.043,E2 -13992.043} C_VEL
LIN {X 0,Y 340.652,Z 341.675,A -85,B 0,C 180,E1 -13996.227,E2 -13996.227} C_VEL
LIN {X 0,Y 340.671,Z 341.67,A -85,B 0,C 180,E1 -13998.688,E2 -13998.688} C_VEL
LIN {X 0,Y 340.721,Z 341.665,A -85,B 0,C 180,E1 -14001.77,E2 -14001.77} C_VEL
LIN {X 0,Y 340.726,Z 341.665,A -85,B 0,C 180,E1 -14005.595,E2 -14005.595} C_VEL
LIN {X 0,Y 340.695,Z 341.671,A -85,B 0,C 180,E1 -14008.954,E2 -14008.954} C_VEL
LIN {X 0,Y 340.712,Z 341.662,A -85,B 0,C 180,E1 -14013.012,E2 -14013.012} C_VEL
LIN {X 0,Y 340.708,Z 341.663,A -85,B 0,C 180,E1 -14016.925,E2 -14016.925} C_VEL
LIN {X 0,Y 340.707,Z 341.649,A -85,B 0,C 180,E1 -14020.728,E2 -14020.728} C_VEL
LIN {X 0,Y 340.796,Z 341.66,A -85,B 0,C 180,E1 -14024.449,E2 -14024.449} C_VEL
LIN {X 0,Y 340.852,Z 341.626,A -85,B 0,C 180,E1 -14028.1,E2 -14028.1} C_VEL
LIN {X 0,Y 340.983,Z 341.626,A -85,B 0,C 180,E1 -14031.704,E2 -14031.704} C_VEL
LIN {X 0,Y 341.019,Z 341.634,A -85,B 0,C 180,E1 -14034.085,E2 -14034.085} C_VEL
LIN {X 0,Y 341.16,Z 341.61,A -85,B 0,C 180,E1 -14037.638,E2 -14037.638} C_VEL
LIN {X 0,Y 341.112,Z 341.611,A -85,B 0,C 180,E1 -14041.18,E2 -14041.18} C_VEL
LIN {X 0,Y 341.129,Z 341.618,A -85,B 0,C 180,E1 -14042.361,E2 -14042.361} C_VEL
LIN {X 0,Y 341.019,Z 341.627,A -85,B 0,C 180,E1 -14045.914,E2 -14045.914} C_VEL
LIN {X 0,Y 340.966,Z 341.637,A -85,B 0,C 180,E1 -14048.356,E2 -14048.356} C_VEL
LIN {X 0,Y 340.852,Z 341.653,A -85,B 0,C 180,E1 -14051.899,E2 -14051.899} C_VEL
LIN {X 0,Y 340.822,Z 341.653,A -85,B 0,C 180,E1 -14055.549,E2 -14055.549} C_VEL
LIN {X 0,Y 340.839,Z 341.65,A -85,B 0,C 180,E1 -14058.466,E2 -14058.466} C_VEL
LIN {X 0,Y 340.756,Z 341.662,A -85,B 0,C 180,E1 -14061.856,E2 -14061.856} C_VEL
LIN {X 0,Y 340.754,Z 341.663,A -85,B 0,C 180,E1 -14065.666,E2 -14065.666} C_VEL
LIN {X 0,Y 340.711,Z 341.668,A -85,B 0,C 180,E1 -14068.322,E2 -14068.322} C_VEL
LIN {X 0,Y 340.697,Z 341.673,A -85,B 0,C 180,E1 -14071.044,E2 -14071.044} C_VEL
LIN {X 0,Y 340.72,Z 341.67,A -85,B 0,C 180,E1 -14075.278,E2 -14075.278} C_VEL
LIN {X 0,Y 340.713,Z 341.667,A -85,B 0,C 180,E1 -14078.386,E2 -14078.386} C_VEL
LIN {X 0,Y 340.7,Z 341.673,A -85,B 0,C 180,E1 -14082.045,E2 -14082.045} C_VEL
LIN {X 0,Y 340.653,Z 341.676,A -85,B 0,C 180,E1 -14086.227,E2 -14086.227} C_VEL
LIN {X 0,Y 340.689,Z 341.673,A -85,B 0,C 180,E1 -14089.753,E2 -14089.753} C_VEL
LIN {X 0,Y 340.706,Z 341.675,A -85,B 0,C 180,E1 -14093.258,E2 -14093.258} C_VEL
LIN {X 0,Y 340.724,Z 341.774,A -85,B 0,C 180,E1 -14096.157,E2 -14096.157} C_VEL
LIN {X 0,Y 343.962,Z 355.334,A -85,B 0,C 180,E1 -14099.724,E2 -14099.724} C_VEL
LIN {X 0,Y 346.051,Z 365.584,A -85,B 0,C 180,E1 -14102.282,E2 -14102.282} C_VEL
LIN {X 0,Y 347.856,Z 371.247,A -85,B 0,C 180,E1 -14102.557,E2 -14102.557} C_VEL
LIN {X 0,Y 352.171,Z 395.954,A -85,B 0,C 180,E1 -14103.431,E2 -14103.431} C_VEL
LIN {X 0,Y 353.874,Z 407.868,A -85,B 0,C 180,E1 -14103.816,E2 -14103.816} C_VEL
LIN {X 0,Y 351.692,Z 503.772,A -85,B 0,C 180,E1 -14105.777,E2 -14105.777} C_VEL
LIN {X 0,Y 350.899,Z 517.682,A -85,B 0,C 180,E1 -14106.268,E2 -14106.268} C_VEL
LIN {X 0,Y 349.755,Z 531.892,A -85,B 0,C 180,E1 -14107.009,E2 -14107.009} C_VEL
LIN {X 0,Y 348.379,Z 545.721,A -85,B 0,C 180,E1 -14107.99,E2 -14107.99} C_VEL
LIN {X 0,Y 347.086,Z 557.772,A -85,B 0,C 180,E1 -14109.091,E2 -14109.091} C_VEL
LIN {X 0,Y 345.561,Z 569.356,A -85,B 0,C 180,E1 -14110.392,E2 -14110.392} C_VEL
LIN {X 0,Y 344.077,Z 579.98,A -85,B 0,C 180,E1 -14111.851,E2 -14111.851} C_VEL
LIN {X 0,Y 342.633,Z 590.532,A -85,B 0,C 180,E1 -14113.618,E2 -14113.618} C_VEL
LIN {X 0,Y 341.551,Z 599.405,A -85,B 0,C 180,E1 -14115.437,E2 -14115.437} C_VEL
LIN {X 0,Y 340.578,Z 607.57,A -85,B 0,C 180,E1 -14117.486,E2 -14117.486} C_VEL
LIN {X 0,Y 339.841,Z 613.38,A -85,B 0,C 180,E1 -14119.273,E2 -14119.273} C_VEL
LIN {X 0,Y 339.465,Z 618.148,A -85,B 0,C 180,E1 -14121.067,E2 -14121.067} C_VEL
LIN {X 0,Y 339.174,Z 623.078,A -85,B 0,C 180,E1 -14123.456,E2 -14123.456} C_VEL
LIN {X 0,Y 339.072,Z 625.765,A -85,B 0,C 180,E1 -14125.244,E2 -14125.244} C_VEL
LIN {X 0,Y 339.005,Z 628.107,A -85,B 0,C 180,E1 -14127.624,E2 -14127.624} C_VEL
LIN {X 0,Y 339.066,Z 629.091,A -85,B 0,C 180,E1 -14130,E2 -14130} C_VEL
LIN {X 0,Y 338.994,Z 628.735,A -85,B 0,C 180,E1 -14132.376,E2 -14132.376} C_VEL
LIN {X 0,Y 339.05,Z 627.046,A -85,B 0,C 180,E1 -14134.756,E2 -14134.756} C_VEL
LIN {X 0,Y 339.251,Z 623.99,A -85,B 0,C 180,E1 -14137.14,E2 -14137.14} C_VEL
LIN {X 0,Y 339.662,Z 619.485,A -85,B 0,C 180,E1 -14139.528,E2 -14139.528} C_VEL
LIN {X 0,Y 340.169,Z 615.032,A -85,B 0,C 180,E1 -14141.319,E2 -14141.319} C_VEL
LIN {X 0,Y 341.258,Z 608.622,A -85,B 0,C 180,E1 -14143.397,E2 -14143.397} C_VEL
LIN {X 0,Y 342.369,Z 600.671,A -85,B 0,C 180,E1 -14145.478,E2 -14145.478} C_VEL
LIN {X 0,Y 343.812,Z 592.376,A -85,B 0,C 180,E1 -14147.242,E2 -14147.242} C_VEL
LIN {X 0,Y 345.556,Z 582.404,A -85,B 0,C 180,E1 -14148.991,E2 -14148.991} C_VEL
LIN {X 0,Y 347.491,Z 571.328,A -85,B 0,C 180,E1 -14150.574,E2 -14150.574} C_VEL
LIN {X 0,Y 349.325,Z 559.258,A -85,B 0,C 180,E1 -14151.973,E2 -14151.973} C_VEL
LIN {X 0,Y 351,Z 546.703,A -85,B 0,C 180,E1 -14153.138,E2 -14153.138} C_VEL
LIN {X 0,Y 352.467,Z 534.204,A -85,B 0,C 180,E1 -14154.049,E2 -14154.049} C_VEL
LIN {X 0,Y 353.861,Z 520.268,A -85,B 0,C 180,E1 -14154.807,E2 -14154.807} C_VEL
LIN {X 0,Y 354.913,Z 505.639,A -85,B 0,C 180,E1 -14155.355,E2 -14155.355} C_VEL
LIN {X 0,Y 355.656,Z 481.485,A -85,B 0,C 180,E1 -14155.891,E2 -14155.891} C_VEL
LIN {X 0,Y 357.449,Z 407.038,A -85,B 0,C 180,E1 -14157.407,E2 -14157.407} C_VEL
LIN {X 0,Y 352.185,Z 379.763,A -85,B 0,C 180,E1 -14158.517,E2 -14158.517} C_VEL
LIN {X 0,Y 351.128,Z 375.793,A -85,B 0,C 180,E1 -14158.71,E2 -14158.71} C_VEL
LIN {X 0,Y 346.557,Z 365.236,A -85,B 0,C 180,E1 -14159.425,E2 -14159.425} C_VEL
LIN {X 0,Y 343.762,Z 353.191,A -85,B 0,C 180,E1 -14162.691,E2 -14162.691} C_VEL
LIN {X 0,Y 340.73,Z 341.668,A -85,B 0,C 180,E1 -14166.059,E2 -14166.059} C_VEL
LIN {X 0,Y 340.7,Z 341.668,A -85,B 0,C 180,E1 -14169.753,E2 -14169.753} C_VEL
LIN {X 0,Y 340.677,Z 341.672,A -85,B 0,C 180,E1 -14172.905,E2 -14172.905} C_VEL
LIN {X 0,Y 340.677,Z 341.672,A -85,B 0,C 180,E1 -14177.096,E2 -14177.096} C_VEL
LIN {X 0,Y 340.701,Z 341.668,A -85,B 0,C 180,E1 -14180.248,E2 -14180.248} C_VEL
LIN {X 0,Y 340.713,Z 341.664,A -85,B 0,C 180,E1 -14183.559,E2 -14183.559} C_VEL
LIN {X 0,Y 340.694,Z 341.669,A -85,B 0,C 180,E1 -14186.154,E2 -14186.154} C_VEL
LIN {X 0,Y 340.725,Z 341.663,A -85,B 0,C 180,E1 -14190.034,E2 -14190.034} C_VEL
LIN {X 0,Y 340.727,Z 341.663,A -85,B 0,C 180,E1 -14193.014,E2 -14193.014} C_VEL
LIN {X 0,Y 340.758,Z 341.663,A -85,B 0,C 180,E1 -14195.639,E2 -14195.639} C_VEL
LIN {X 0,Y 340.74,Z 341.663,A -85,B 0,C 180,E1 -14199.474,E2 -14199.474} C_VEL
LIN {X 0,Y 340.861,Z 341.643,A -85,B 0,C 180,E1 -14201.985,E2 -14201.985} C_VEL
LIN {X 0,Y 340.872,Z 341.647,A -85,B 0,C 180,E1 -14205.705,E2 -14205.705} C_VEL
LIN {X 0,Y 340.873,Z 341.648,A -85,B 0,C 180,E1 -14209.307,E2 -14209.307} C_VEL
LIN {X 0,Y 341.006,Z 341.628,A -85,B 0,C 180,E1 -14212.897,E2 -14212.897} C_VEL
LIN {X 0,Y 340.82,Z 341.654,A -85,B 0,C 180,E1 -14215.269,E2 -14215.269} C_VEL
LIN {X 0,Y 341.129,Z 341.609,A -85,B 0,C 180,E1 -14217.639,E2 -14217.639} C_VEL
LIN {X 0,Y 341.092,Z 341.615,A -85,B 0,C 180,E1 -14221.181,E2 -14221.181} C_VEL
LIN {X 0,Y 341.16,Z 341.606,A -85,B 0,C 180,E1 -14222.362,E2 -14222.362} C_VEL
LIN {X 0,Y 341.005,Z 341.62,A -85,B 0,C 180,E1 -14227.104,E2 -14227.104} C_VEL
LIN {X 0,Y 340.851,Z 341.647,A -85,B 0,C 180,E1 -14230.695,E2 -14230.695} C_VEL
LIN {X 0,Y 340.821,Z 341.655,A -85,B 0,C 180,E1 -14234.327,E2 -14234.327} C_VEL
LIN {X 0,Y 340.758,Z 341.663,A -85,B 0,C 180,E1 -14238.425,E2 -14238.425} C_VEL
LIN {X 0,Y 340.721,Z 341.666,A -85,B 0,C 180,E1 -14241.842,E2 -14241.842} C_VEL
LIN {X 0,Y 340.673,Z 341.67,A -85,B 0,C 180,E1 -14245.673,E2 -14245.673} C_VEL
LIN {X 0,Y 340.678,Z 341.666,A -85,B 0,C 180,E1 -14248.326,E2 -14248.326} C_VEL
LIN {X 0,Y 340.685,Z 341.647,A -85,B 0,C 180,E1 -14251.046,E2 -14251.046} C_VEL
LIN {X 0,Y 340.718,Z 341.656,A -85,B 0,C 180,E1 -14255.279,E2 -14255.279} C_VEL
LIN {X 0,Y 340.696,Z 341.669,A -85,B 0,C 180,E1 -14258.382,E2 -14258.382} C_VEL
LIN {X 0,Y 340.693,Z 341.671,A -85,B 0,C 180,E1 -14262.044,E2 -14262.044} C_VEL
LIN {X 0,Y 340.652,Z 341.668,A -85,B 0,C 180,E1 -14266.228,E2 -14266.228} C_VEL
LIN {X 0,Y 340.671,Z 341.672,A -85,B 0,C 180,E1 -14268.688,E2 -14268.688} C_VEL
LIN {X 0,Y 340.722,Z 341.672,A -85,B 0,C 180,E1 -14272.519,E2 -14272.519} C_VEL
LIN {X 0,Y 340.742,Z 341.787,A -85,B 0,C 180,E1 -14272.939,E2 -14272.939} C_VEL
LIN {X 0,Y 342.652,Z 349.273,A -85,B 0,C 180,E1 -14275.249,E2 -14275.249} C_VEL
LIN {X 0,Y 351.283,Z 367.174,A -85,B 0,C 180,E1 -14276.543,E2 -14276.543} C_VEL
LIN {X 0,Y 358.019,Z 382.971,A -85,B 0,C 180,E1 -14277.539,E2 -14277.539} C_VEL
LIN {X 0,Y 355.486,Z 485.145,A -85,B 0,C 180,E1 -14279.644,E2 -14279.644} C_VEL
LIN {X 0,Y 354.684,Z 499.26,A -85,B 0,C 180,E1 -14280.142,E2 -14280.142} C_VEL
LIN {X 0,Y 353.505,Z 512.638,A -85,B 0,C 180,E1 -14280.826,E2 -14280.826} C_VEL
LIN {X 0,Y 352.16,Z 525.413,A -85,B 0,C 180,E1 -14281.707,E2 -14281.707} C_VEL
LIN {X 0,Y 350.533,Z 538.402,A -85,B 0,C 180,E1 -14282.862,E2 -14282.862} C_VEL
LIN {X 0,Y 348.758,Z 550.15,A -85,B 0,C 180,E1 -14284.165,E2 -14284.165} C_VEL
LIN {X 0,Y 347.051,Z 561.211,A -85,B 0,C 180,E1 -14285.684,E2 -14285.684} C_VEL
LIN {X 0,Y 345.414,Z 570.671,A -85,B 0,C 180,E1 -14287.258,E2 -14287.258} C_VEL
LIN {X 0,Y 343.824,Z 579.531,A -85,B 0,C 180,E1 -14289.04,E2 -14289.04} C_VEL
LIN {X 0,Y 342.532,Z 586.875,A -85,B 0,C 180,E1 -14290.835,E2 -14290.835} C_VEL
LIN {X 0,Y 341.499,Z 592.968,A -85,B 0,C 180,E1 -14292.638,E2 -14292.638} C_VEL
LIN {X 0,Y 340.441,Z 599.42,A -85,B 0,C 180,E1 -14295.046,E2 -14295.046} C_VEL
LIN {X 0,Y 339.673,Z 604.216,A -85,B 0,C 180,E1 -14297.452,E2 -14297.452} C_VEL
LIN {X 0,Y 339.276,Z 606.785,A -85,B 0,C 180,E1 -14299.255,E2 -14299.255} C_VEL
LIN {X 0,Y 339.1,Z 609.002,A -85,B 0,C 180,E1 -14301.658,E2 -14301.658} C_VEL
LIN {X 0,Y 339.114,Z 609.874,A -85,B 0,C 180,E1 -14304.052,E2 -14304.052} C_VEL
LIN {X 0,Y 339.071,Z 609.433,A -85,B 0,C 180,E1 -14306.435,E2 -14306.435} C_VEL
LIN {X 0,Y 339.096,Z 607.676,A -85,B 0,C 180,E1 -14308.812,E2 -14308.812} C_VEL
LIN {X 0,Y 339.328,Z 604.567,A -85,B 0,C 180,E1 -14311.187,E2 -14311.187} C_VEL
LIN {X 0,Y 339.776,Z 599.996,A -85,B 0,C 180,E1 -14313.558,E2 -14313.558} C_VEL
LIN {X 0,Y 340.454,Z 595.501,A -85,B 0,C 180,E1 -14315.33,E2 -14315.33} C_VEL
LIN {X 0,Y 341.19,Z 589.034,A -85,B 0,C 180,E1 -14317.397,E2 -14317.397} C_VEL
LIN {X 0,Y 342.258,Z 581.019,A -85,B 0,C 180,E1 -14319.455,E2 -14319.455} C_VEL
LIN {X 0,Y 343.336,Z 572.636,A -85,B 0,C 180,E1 -14321.213,E2 -14321.213} C_VEL
LIN {X 0,Y 344.883,Z 562.497,A -85,B 0,C 180,E1 -14322.953,E2 -14322.953} C_VEL
LIN {X 0,Y 346.295,Z 551.172,A -85,B 0,C 180,E1 -14324.546,E2 -14324.546} C_VEL
LIN {X 0,Y 347.668,Z 539.897,A -85,B 0,C 180,E1 -14325.837,E2 -14325.837} C_VEL
LIN {X 0,Y 349.024,Z 527.568,A -85,B 0,C 180,E1 -14326.976,E2 -14326.976} C_VEL
LIN {X 0,Y 350.257,Z 513.815,A -85,B 0,C 180,E1 -14327.969,E2 -14327.969} C_VEL
LIN {X 0,Y 351.272,Z 499.963,A -85,B 0,C 180,E1 -14328.708,E2 -14328.708} C_VEL
LIN {X 0,Y 351.959,Z 485.505,A -85,B 0,C 180,E1 -14329.237,E2 -14329.237} C_VEL
LIN {X 0,Y 353.26,Z 430.089,A -85,B 0,C 180,E1 -14330.383,E2 -14330.383} C_VEL
LIN {X 0,Y 352.807,Z 424.284,A -85,B 0,C 180,E1 -14330.542,E2 -14330.542} C_VEL
LIN {X 0,Y 348.04,Z 405.6,A -85,B 0,C 180,E1 -14331.302,E2 -14331.302} C_VEL
LIN {X 0,Y 347.538,Z 399.796,A -85,B 0,C 180,E1 -14331.469,E2 -14331.469} C_VEL
LIN {X 0,Y 347.812,Z 382.251,A -85,B 0,C 180,E1 -14331.839,E2 -14331.839} C_VEL
LIN {X 0,Y 346.543,Z 377.026,A -85,B 0,C 180,E1 -14332.055,E2 -14332.055} C_VEL
LIN {X 0,Y 338.678,Z 357.226,A -85,B 0,C 180,E1 -14333.141,E2 -14333.141} C_VEL
LIN {X 0,Y 335.19,Z 348.96,A -85,B 0,C 180,E1 -14333.641,E2 -14333.641} C_VEL
LIN {X 0,Y 333.628,Z 342.556,A -85,B 0,C 180,E1 -14335.607,E2 -14335.607} C_VEL
LIN {X 0,Y 333.651,Z 342.55,A -85,B 0,C 180,E1 -14338.978,E2 -14338.978} C_VEL
LIN {X 0,Y 333.642,Z 342.55,A -85,B 0,C 180,E1 -14342.586,E2 -14342.586} C_VEL
LIN {X 0,Y 333.676,Z 342.546,A -85,B 0,C 180,E1 -14346.139,E2 -14346.139} C_VEL
LIN {X 0,Y 333.604,Z 342.552,A -85,B 0,C 180,E1 -14349.199,E2 -14349.199} C_VEL
LIN {X 0,Y 333.629,Z 342.549,A -85,B 0,C 180,E1 -14352.498,E2 -14352.498} C_VEL
LIN {X 0,Y 333.596,Z 342.552,A -85,B 0,C 180,E1 -14355.954,E2 -14355.954} C_VEL
LIN {X 0,Y 333.604,Z 342.552,A -85,B 0,C 180,E1 -14359.324,E2 -14359.324} C_VEL
LIN {X 0,Y 333.665,Z 342.543,A -85,B 0,C 180,E1 -14363.168,E2 -14363.168} C_VEL
LIN {X 0,Y 333.677,Z 342.544,A -85,B 0,C 180,E1 -14365.341,E2 -14365.341} C_VEL
LIN {X 0,Y 333.631,Z 342.544,A -85,B 0,C 180,E1 -14368.221,E2 -14368.221} C_VEL
LIN {X 0,Y 333.631,Z 342.547,A -85,B 0,C 180,E1 -14371.02,E2 -14371.02} C_VEL
LIN {X 0,Y 333.66,Z 342.547,A -85,B 0,C 180,E1 -14374.922,E2 -14374.922} C_VEL
LIN {X 0,Y 333.654,Z 342.523,A -85,B 0,C 180,E1 -14379.017,E2 -14379.017} C_VEL
LIN {X 0,Y 333.714,Z 342.527,A -85,B 0,C 180,E1 -14381.584,E2 -14381.584} C_VEL
LIN {X 0,Y 333.776,Z 342.531,A -85,B 0,C 180,E1 -14385.6,E2 -14385.6} C_VEL
LIN {X 0,Y 333.82,Z 342.495,A -85,B 0,C 180,E1 -14389.077,E2 -14389.077} C_VEL
LIN {X 0,Y 333.96,Z 342.509,A -85,B 0,C 180,E1 -14392.746,E2 -14392.746} C_VEL
LIN {X 0,Y 333.792,Z 342.527,A -85,B 0,C 180,E1 -14395.168,E2 -14395.168} C_VEL
LIN {X 0,Y 334.096,Z 342.49,A -85,B 0,C 180,E1 -14397.588,E2 -14397.588} C_VEL
LIN {X 0,Y 334.081,Z 342.486,A -85,B 0,C 180,E1 -14401.205,E2 -14401.205} C_VEL
LIN {X 0,Y 333.81,Z 342.529,A -85,B 0,C 180,E1 -14403.621,E2 -14403.621} C_VEL
LIN {X 0,Y 333.993,Z 342.502,A -85,B 0,C 180,E1 -14406.039,E2 -14406.039} C_VEL
LIN {X 0,Y 333.823,Z 342.525,A -85,B 0,C 180,E1 -14409.696,E2 -14409.696} C_VEL
LIN {X 0,Y 333.799,Z 342.529,A -85,B 0,C 180,E1 -14413.391,E2 -14413.391} C_VEL
LIN {X 0,Y 333.749,Z 342.535,A -85,B 0,C 180,E1 -14417.146,E2 -14417.146} C_VEL
LIN {X 0,Y 333.737,Z 342.538,A -85,B 0,C 180,E1 -14419.69,E2 -14419.69} C_VEL
LIN {X 0,Y 333.694,Z 342.541,A -85,B 0,C 180,E1 -14422.278,E2 -14422.278} C_VEL
LIN {X 0,Y 333.71,Z 342.54,A -85,B 0,C 180,E1 -14425.097,E2 -14425.097} C_VEL
LIN {X 0,Y 333.679,Z 342.543,A -85,B 0,C 180,E1 -14428.975,E2 -14428.975} C_VEL
LIN {X 0,Y 333.64,Z 342.549,A -85,B 0,C 180,E1 -14433.208,E2 -14433.208} C_VEL
LIN {X 0,Y 333.668,Z 342.548,A -85,B 0,C 180,E1 -14436.832,E2 -14436.832} C_VEL
LIN {X 0,Y 333.648,Z 342.55,A -85,B 0,C 180,E1 -14440.767,E2 -14440.767} C_VEL
LIN {X 0,Y 333.594,Z 342.556,A -85,B 0,C 180,E1 -14444.25,E2 -14444.25} C_VEL
LIN {X 0,Y 333.642,Z 342.55,A -85,B 0,C 180,E1 -14447.618,E2 -14447.618} C_VEL
LIN {X 0,Y 333.654,Z 342.553,A -85,B 0,C 180,E1 -14451.202,E2 -14451.202} C_VEL
LIN {X 0,Y 333.677,Z 342.554,A -85,B 0,C 180,E1 -14453.861,E2 -14453.861} C_VEL
LIN {X 0,Y 333.687,Z 342.589,A -85,B 0,C 180,E1 -14455.663,E2 -14455.663} C_VEL
LIN {X 0,Y 336.981,Z 356.325,A -85,B 0,C 180,E1 -14459.376,E2 -14459.376} C_VEL
LIN {X 0,Y 338.826,Z 365.449,A -85,B 0,C 180,E1 -14461.701,E2 -14461.701} C_VEL
LIN {X 0,Y 341.691,Z 373.551,A -85,B 0,C 180,E1 -14462.121,E2 -14462.121} C_VEL
LIN {X 0,Y 346.137,Z 399.924,A -85,B 0,C 180,E1 -14463.067,E2 -14463.067} C_VEL
LIN {X 0,Y 347.392,Z 408.819,A -85,B 0,C 180,E1 -14463.36,E2 -14463.36} C_VEL
LIN {X 0,Y 345.152,Z 503.441,A -85,B 0,C 180,E1 -14465.328,E2 -14465.328} C_VEL
LIN {X 0,Y 344.277,Z 518.164,A -85,B 0,C 180,E1 -14465.863,E2 -14465.863} C_VEL
LIN {X 0,Y 343.084,Z 532.196,A -85,B 0,C 180,E1 -14466.616,E2 -14466.616} C_VEL
LIN {X 0,Y 341.667,Z 545.745,A -85,B 0,C 180,E1 -14467.599,E2 -14467.599} C_VEL
LIN {X 0,Y 340.245,Z 558.611,A -85,B 0,C 180,E1 -14468.809,E2 -14468.809} C_VEL
LIN {X 0,Y 338.665,Z 570.011,A -85,B 0,C 180,E1 -14470.134,E2 -14470.134} C_VEL
LIN {X 0,Y 336.997,Z 581.464,A -85,B 0,C 180,E1 -14471.771,E2 -14471.771} C_VEL
LIN {X 0,Y 335.533,Z 591.678,A -85,B 0,C 180,E1 -14473.574,E2 -14473.574} C_VEL
LIN {X 0,Y 334.479,Z 600.158,A -85,B 0,C 180,E1 -14475.396,E2 -14475.396} C_VEL
LIN {X 0,Y 333.446,Z 608.246,A -85,B 0,C 180,E1 -14477.524,E2 -14477.524} C_VEL
LIN {X 0,Y 332.665,Z 614.755,A -85,B 0,C 180,E1 -14479.655,E2 -14479.655} C_VEL
LIN {X 0,Y 332.212,Z 620.524,A -85,B 0,C 180,E1 -14482.096,E2 -14482.096} C_VEL
LIN {X 0,Y 332.062,Z 624.096,A -85,B 0,C 180,E1 -14484.121,E2 -14484.121} C_VEL
LIN {X 0,Y 331.99,Z 626.871,A -85,B 0,C 180,E1 -14486.359,E2 -14486.359} C_VEL
LIN {X 0,Y 331.926,Z 628.549,A -85,B 0,C 180,E1 -14488.787,E2 -14488.787} C_VEL
LIN {X 0,Y 331.969,Z 628.884,A -85,B 0,C 180,E1 -14490,E2 -14490} C_VEL
LIN {X 0,Y 331.911,Z 628.55,A -85,B 0,C 180,E1 -14492.427,E2 -14492.427} C_VEL
LIN {X 0,Y 331.959,Z 626.882,A -85,B 0,C 180,E1 -14494.858,E2 -14494.858} C_VEL
LIN {X 0,Y 332.175,Z 623.848,A -85,B 0,C 180,E1 -14497.293,E2 -14497.293} C_VEL
LIN {X 0,Y 332.621,Z 619.367,A -85,B 0,C 180,E1 -14499.732,E2 -14499.732} C_VEL
LIN {X 0,Y 333.185,Z 614.94,A -85,B 0,C 180,E1 -14501.56,E2 -14501.56} C_VEL
LIN {X 0,Y 334.302,Z 608.557,A -85,B 0,C 180,E1 -14503.681,E2 -14503.681} C_VEL
LIN {X 0,Y 335.505,Z 600.638,A -85,B 0,C 180,E1 -14505.802,E2 -14505.802} C_VEL
LIN {X 0,Y 337.017,Z 592.378,A -85,B 0,C 180,E1 -14507.601,E2 -14507.601} C_VEL
LIN {X 0,Y 338.829,Z 582.449,A -85,B 0,C 180,E1 -14509.383,E2 -14509.383} C_VEL
LIN {X 0,Y 340.85,Z 571.425,A -85,B 0,C 180,E1 -14510.993,E2 -14510.993} C_VEL
LIN {X 0,Y 342.796,Z 559.133,A -85,B 0,C 180,E1 -14512.449,E2 -14512.449} C_VEL
LIN {X 0,Y 344.489,Z 546.992,A -85,B 0,C 180,E1 -14513.601,E2 -14513.601} C_VEL
LIN {X 0,Y 346.008,Z 534.631,A -85,B 0,C 180,E1 -14514.527,E2 -14514.527} C_VEL
LIN {X 0,Y 347.468,Z 520.913,A -85,B 0,C 180,E1 -14515.295,E2 -14515.295} C_VEL
LIN {X 0,Y 348.551,Z 506.706,A -85,B 0,C 180,E1 -14515.851,E2 -14515.851} C_VEL
LIN {X 0,Y 349.235,Z 487.392,A -85,B 0,C 180,E1 -14516.31,E2 -14516.31} C_VEL
LIN {X 0,Y 351.271,Z 408.316,A -85,B 0,C 180,E1 -14517.942,E2 -14517.942} C_VEL
LIN {X 0,Y 346.052,Z 381.155,A -85,B 0,C 180,E1 -14519.08,E2 -14519.08} C_VEL
LIN {X 0,Y 345.043,Z 377.962,A -85,B 0,C 180,E1 -14519.256,E2 -14519.256} C_VEL
LIN {X 0,Y 339.306,Z 364.922,A -85,B 0,C 180,E1 -14520.196,E2 -14520.196} C_VEL
LIN {X 0,Y 336.612,Z 353.61,A -85,B 0,C 180,E1 -14523.369,E2 -14523.369} C_VEL
LIN {X 0,Y 333.681,Z 342.546,A -85,B 0,C 180,E1 -14526.685,E2 -14526.685} C_VEL
LIN {X 0,Y 333.648,Z 342.55,A -85,B 0,C 180,E1 -14530.685,E2 -14530.685} C_VEL
LIN {X 0,Y 333.594,Z 342.556,A -85,B 0,C 180,E1 -14534.251,E2 -14534.251} C_VEL
LIN {X 0,Y 333.643,Z 342.548,A -85,B 0,C 180,E1 -14537.619,E2 -14537.619} C_VEL
LIN {X 0,Y 333.655,Z 342.544,A -85,B 0,C 180,E1 -14541.202,E2 -14541.202} C_VEL
LIN {X 0,Y 333.679,Z 342.54,A -85,B 0,C 180,E1 -14543.862,E2 -14543.862} C_VEL
LIN {X 0,Y 333.645,Z 342.545,A -85,B 0,C 180,E1 -14547.413,E2 -14547.413} C_VEL
LIN {X 0,Y 333.657,Z 342.546,A -85,B 0,C 180,E1 -14551.023,E2 -14551.023} C_VEL
LIN {X 0,Y 333.711,Z 342.539,A -85,B 0,C 180,E1 -14555.09,E2 -14555.09} C_VEL
LIN {X 0,Y 333.678,Z 342.543,A -85,B 0,C 180,E1 -14559.019,E2 -14559.019} C_VEL
LIN {X 0,Y 333.797,Z 342.525,A -85,B 0,C 180,E1 -14561.59,E2 -14561.59} C_VEL
LIN {X 0,Y 333.811,Z 342.528,A -85,B 0,C 180,E1 -14565.577,E2 -14565.577} C_VEL
LIN {X 0,Y 333.836,Z 342.524,A -85,B 0,C 180,E1 -14569.078,E2 -14569.078} C_VEL
LIN {X 0,Y 333.961,Z 342.506,A -85,B 0,C 180,E1 -14572.746,E2 -14572.746} C_VEL
LIN {X 0,Y 333.786,Z 342.53,A -85,B 0,C 180,E1 -14575.169,E2 -14575.169} C_VEL
LIN {X 0,Y 334.07,Z 342.487,A -85,B 0,C 180,E1 -14577.589,E2 -14577.589} C_VEL
LIN {X 0,Y 334.063,Z 342.49,A -85,B 0,C 180,E1 -14581.206,E2 -14581.206} C_VEL
LIN {X 0,Y 334.097,Z 342.486,A -85,B 0,C 180,E1 -14582.412,E2 -14582.412} C_VEL
LIN {X 0,Y 333.964,Z 342.497,A -85,B 0,C 180,E1 -14586.46,E2 -14586.46} C_VEL
LIN {X 0,Y 333.824,Z 342.529,A -85,B 0,C 180,E1 -14589.697,E2 -14589.697} C_VEL
LIN {X 0,Y 333.79,Z 342.529,A -85,B 0,C 180,E1 -14593.392,E2 -14593.392} C_VEL
LIN {X 0,Y 333.683,Z 342.537,A -85,B 0,C 180,E1 -14597.15,E2 -14597.15} C_VEL
LIN {X 0,Y 333.639,Z 342.546,A -85,B 0,C 180,E1 -14599.697,E2 -14599.697} C_VEL
LIN {X 0,Y 333.653,Z 342.548,A -85,B 0,C 180,E1 -14602.281,E2 -14602.281} C_VEL
LIN {X 0,Y 333.661,Z 342.54,A -85,B 0,C 180,E1 -14605.078,E2 -14605.078} C_VEL
LIN {X 0,Y 333.631,Z 342.533,A -85,B 0,C 180,E1 -14608.98,E2 -14608.98} C_VEL
LIN {X 0,Y 333.643,Z 342.546,A -85,B 0,C 180,E1 -14612.586,E2 -14612.586} C_VEL
LIN {X 0,Y 333.676,Z 342.524,A -85,B 0,C 180,E1 -14616.14,E2 -14616.14} C_VEL
LIN {X 0,Y 333.623,Z 342.554,A -85,B 0,C 180,E1 -14619.196,E2 -14619.196} C_VEL
LIN {X 0,Y 333.629,Z 342.55,A -85,B 0,C 180,E1 -14622.499,E2 -14622.499} C_VEL
LIN {X 0,Y 333.596,Z 342.546,A -85,B 0,C 180,E1 -14625.954,E2 -14625.954} C_VEL
LIN {X 0,Y 333.604,Z 342.549,A -85,B 0,C 180,E1 -14629.325,E2 -14629.325} C_VEL
LIN {X 0,Y 333.687,Z 342.657,A -85,B 0,C 180,E1 -14632.306,E2 -14632.306} C_VEL
LIN {X 0,Y 335.484,Z 349.466,A -85,B 0,C 180,E1 -14634.484,E2 -14634.484} C_VEL
LIN {X 0,Y 344.54,Z 367.998,A -85,B 0,C 180,E1 -14635.894,E2 -14635.894} C_VEL
LIN {X 0,Y 351.895,Z 385.023,A -85,B 0,C 180,E1 -14637.016,E2 -14637.016} C_VEL
LIN {X 0,Y 349.196,Z 485.756,A -85,B 0,C 180,E1 -14639.121,E2 -14639.121} C_VEL
LIN {X 0,Y 348.288,Z 500.483,A -85,B 0,C 180,E1 -14639.662,E2 -14639.662} C_VEL
LIN {X 0,Y 347.008,Z 514.167,A -85,B 0,C 180,E1 -14640.393,E2 -14640.393} C_VEL
LIN {X 0,Y 345.589,Z 527.061,A -85,B 0,C 180,E1 -14641.323,E2 -14641.323} C_VEL
LIN {X 0,Y 343.936,Z 539.437,A -85,B 0,C 180,E1 -14642.463,E2 -14642.463} C_VEL
LIN {X 0,Y 342.089,Z 551.036,A -85,B 0,C 180,E1 -14643.787,E2 -14643.787} C_VEL
LIN {X 0,Y 340.342,Z 561.844,A -85,B 0,C 180,E1 -14645.313,E2 -14645.313} C_VEL
LIN {X 0,Y 338.482,Z 572.165,A -85,B 0,C 180,E1 -14647.088,E2 -14647.088} C_VEL
LIN {X 0,Y 336.822,Z 580.806,A -85,B 0,C 180,E1 -14648.904,E2 -14648.904} C_VEL
LIN {X 0,Y 335.327,Z 589.043,A -85,B 0,C 180,E1 -14651.043,E2 -14651.043} C_VEL
LIN {X 0,Y 334.252,Z 594.79,A -85,B 0,C 180,E1 -14652.88,E2 -14652.88} C_VEL
LIN {X 0,Y 333.486,Z 599.471,A -85,B 0,C 180,E1 -14654.726,E2 -14654.726} C_VEL
LIN {X 0,Y 332.664,Z 604.305,A -85,B 0,C 180,E1 -14657.183,E2 -14657.183} C_VEL
LIN {X 0,Y 332.234,Z 606.91,A -85,B 0,C 180,E1 -14659.025,E2 -14659.025} C_VEL
LIN {X 0,Y 332.013,Z 609.162,A -85,B 0,C 180,E1 -14661.479,E2 -14661.479} C_VEL
LIN {X 0,Y 332.032,Z 610.068,A -85,B 0,C 180,E1 -14663.925,E2 -14663.925} C_VEL
LIN {X 0,Y 331.995,Z 609.659,A -85,B 0,C 180,E1 -14666.359,E2 -14666.359} C_VEL
LIN {X 0,Y 331.998,Z 607.937,A -85,B 0,C 180,E1 -14668.787,E2 -14668.787} C_VEL
LIN {X 0,Y 332.236,Z 604.863,A -85,B 0,C 180,E1 -14671.212,E2 -14671.212} C_VEL
LIN {X 0,Y 332.7,Z 600.345,A -85,B 0,C 180,E1 -14673.633,E2 -14673.633} C_VEL
LIN {X 0,Y 333.415,Z 595.871,A -85,B 0,C 180,E1 -14675.443,E2 -14675.443} C_VEL
LIN {X 0,Y 334.177,Z 589.448,A -85,B 0,C 180,E1 -14677.553,E2 -14677.553} C_VEL
LIN {X 0,Y 335.27,Z 581.483,A -85,B 0,C 180,E1 -14679.654,E2 -14679.654} C_VEL
LIN {X 0,Y 336.414,Z 573.149,A -85,B 0,C 180,E1 -14681.447,E2 -14681.447} C_VEL
LIN {X 0,Y 338.003,Z 563.098,A -85,B 0,C 180,E1 -14683.222,E2 -14683.222} C_VEL
LIN {X 0,Y 339.475,Z 551.863,A -85,B 0,C 180,E1 -14684.844,E2 -14684.844} C_VEL
LIN {X 0,Y 340.881,Z 540.694,A -85,B 0,C 180,E1 -14686.161,E2 -14686.161} C_VEL
LIN {X 0,Y 342.285,Z 528.506,A -85,B 0,C 180,E1 -14687.321,E2 -14687.321} C_VEL
LIN {X 0,Y 343.548,Z 514.961,A -85,B 0,C 180,E1 -14688.332,E2 -14688.332} C_VEL
LIN {X 0,Y 344.668,Z 500.679,A -85,B 0,C 180,E1 -14689.119,E2 -14689.119} C_VEL
LIN {X 0,Y 345.344,Z 486.488,A -85,B 0,C 180,E1 -14689.659,E2 -14689.659} C_VEL
LIN {X 0,Y 346.579,Z 437.773,A -85,B 0,C 180,E1 -14690.695,E2 -14690.695} C_VEL
LIN {X 0,Y 347.538,Z 399.796,A -85,B 0,C 180,E1 -14691.469,E2 -14691.469} C_VEL
LIN {X 0,Y 346.963,Z 393.98,A -85,B 0,C 180,E1 -14691.642,E2 -14691.642} C_VEL
LIN {X 0,Y 345.366,Z 388.42,A -85,B 0,C 180,E1 -14691.89,E2 -14691.89} C_VEL
LIN {X 0,Y 340.516,Z 377.905,A -85,B 0,C 180,E1 -14692.513,E2 -14692.513} C_VEL
LIN {X 0,Y 337.105,Z 370.946,A -85,B 0,C 180,E1 -14692.953,E2 -14692.953} C_VEL
LIN {X 0,Y 329.3,Z 352.215,A -85,B 0,C 180,E1 -14694.069,E2 -14694.069} C_VEL
LIN {X 0,Y 327.987,Z 349.156,A -85,B 0,C 180,E1 -14694.278,E2 -14694.278} C_VEL
LIN {X 0,Y 326.599,Z 343.433,A -85,B 0,C 180,E1 -14696.081,E2 -14696.081} C_VEL
LIN {X 0,Y 326.59,Z 343.423,A -85,B 0,C 180,E1 -14699.666,E2 -14699.666} C_VEL
LIN {X 0,Y 326.617,Z 343.425,A -85,B 0,C 180,E1 -14702.945,E2 -14702.945} C_VEL
LIN {X 0,Y 326.613,Z 343.425,A -85,B 0,C 180,E1 -14705.52,E2 -14705.52} C_VEL
LIN {X 0,Y 326.574,Z 343.428,A -85,B 0,C 180,E1 -14709.218,E2 -14709.218} C_VEL
LIN {X 0,Y 326.574,Z 343.432,A -85,B 0,C 180,E1 -14712.971,E2 -14712.971} C_VEL
LIN {X 0,Y 326.574,Z 343.43,A -85,B 0,C 180,E1 -14717.029,E2 -14717.029} C_VEL
LIN {X 0,Y 326.589,Z 343.43,A -85,B 0,C 180,E1 -14720.778,E2 -14720.778} C_VEL
LIN {X 0,Y 326.615,Z 343.426,A -85,B 0,C 180,E1 -14724.48,E2 -14724.48} C_VEL
LIN {X 0,Y 326.611,Z 343.415,A -85,B 0,C 180,E1 -14727.455,E2 -14727.455} C_VEL
LIN {X 0,Y 326.582,Z 343.431,A -85,B 0,C 180,E1 -14730.333,E2 -14730.333} C_VEL
LIN {X 0,Y 326.598,Z 343.42,A -85,B 0,C 180,E1 -14733.134,E2 -14733.134} C_VEL
LIN {X 0,Y 326.614,Z 343.425,A -85,B 0,C 180,E1 -14735.868,E2 -14735.868} C_VEL
LIN {X 0,Y 326.611,Z 343.404,A -85,B 0,C 180,E1 -14738.542,E2 -14738.542} C_VEL
LIN {X 0,Y 326.65,Z 343.406,A -85,B 0,C 180,E1 -14741.206,E2 -14741.206} C_VEL
LIN {X 0,Y 326.728,Z 343.408,A -85,B 0,C 180,E1 -14745.459,E2 -14745.459} C_VEL
LIN {X 0,Y 326.761,Z 343.374,A -85,B 0,C 180,E1 -14748.838,E2 -14748.838} C_VEL
LIN {X 0,Y 326.917,Z 343.387,A -85,B 0,C 180,E1 -14752.589,E2 -14752.589} C_VEL
LIN {X 0,Y 326.76,Z 343.403,A -85,B 0,C 180,E1 -14755.064,E2 -14755.064} C_VEL
LIN {X 0,Y 327.037,Z 343.369,A -85,B 0,C 180,E1 -14757.536,E2 -14757.536} C_VEL
LIN {X 0,Y 327.049,Z 343.362,A -85,B 0,C 180,E1 -14761.231,E2 -14761.231} C_VEL
LIN {X 0,Y 326.759,Z 343.408,A -85,B 0,C 180,E1 -14763.699,E2 -14763.699} C_VEL
LIN {X 0,Y 326.947,Z 343.38,A -85,B 0,C 180,E1 -14766.17,E2 -14766.17} C_VEL
LIN {X 0,Y 326.786,Z 343.4,A -85,B 0,C 180,E1 -14769.907,E2 -14769.907} C_VEL
LIN {X 0,Y 326.762,Z 343.405,A -85,B 0,C 180,E1 -14773.685,E2 -14773.685} C_VEL
LIN {X 0,Y 326.702,Z 343.414,A -85,B 0,C 180,E1 -14777.527,E2 -14777.527} C_VEL
LIN {X 0,Y 326.664,Z 343.42,A -85,B 0,C 180,E1 -14780.135,E2 -14780.135} C_VEL
LIN {X 0,Y 326.648,Z 343.422,A -85,B 0,C 180,E1 -14784.129,E2 -14784.129} C_VEL
LIN {X 0,Y 326.64,Z 343.422,A -85,B 0,C 180,E1 -14788.252,E2 -14788.252} C_VEL
LIN {X 0,Y 326.577,Z 343.432,A -85,B 0,C 180,E1 -14791.097,E2 -14791.097} C_VEL
LIN {X 0,Y 326.609,Z 343.43,A -85,B 0,C 180,E1 -14794.019,E2 -14794.019} C_VEL
LIN {X 0,Y 326.631,Z 343.427,A -85,B 0,C 180,E1 -14797.239,E2 -14797.239} C_VEL
LIN {X 0,Y 326.579,Z 343.432,A -85,B 0,C 180,E1 -14801.131,E2 -14801.131} C_VEL
LIN {X 0,Y 326.528,Z 343.437,A -85,B 0,C 180,E1 -14804.743,E2 -14804.743} C_VEL
LIN {X 0,Y 326.577,Z 343.429,A -85,B 0,C 180,E1 -14808.154,E2 -14808.154} C_VEL
LIN {X 0,Y 326.624,Z 343.428,A -85,B 0,C 180,E1 -14811.391,E2 -14811.391} C_VEL
LIN {X 0,Y 326.664,Z 343.486,A -85,B 0,C 180,E1 -14815.17,E2 -14815.17} C_VEL
LIN {X 0,Y 329.761,Z 356.557,A -85,B 0,C 180,E1 -14818.802,E2 -14818.802} C_VEL
LIN {X 0,Y 331.649,Z 365.281,A -85,B 0,C 180,E1 -14821.089,E2 -14821.089} C_VEL
LIN {X 0,Y 335.412,Z 375.34,A -85,B 0,C 180,E1 -14821.647,E2 -14821.647} C_VEL
LIN {X 0,Y 339.841,Z 401.714,A -85,B 0,C 180,E1 -14822.618,E2 -14822.618} C_VEL
LIN {X 0,Y 340.951,Z 409.002,A -85,B 0,C 180,E1 -14822.871,E2 -14822.871} C_VEL
LIN {X 0,Y 338.634,Z 503.092,A -85,B 0,C 180,E1 -14824.861,E2 -14824.861} C_VEL
LIN {X 0,Y 337.708,Z 517.868,A -85,B 0,C 180,E1 -14825.404,E2 -14825.404} C_VEL
LIN {X 0,Y 336.524,Z 531.355,A -85,B 0,C 180,E1 -14826.132,E2 -14826.132} C_VEL
LIN {X 0,Y 335.015,Z 545.431,A -85,B 0,C 180,E1 -14827.164,E2 -14827.164} C_VEL
LIN {X 0,Y 333.569,Z 558.007,A -85,B 0,C 180,E1 -14828.364,E2 -14828.364} C_VEL
LIN {X 0,Y 331.774,Z 570.66,A -85,B 0,C 180,E1 -14829.865,E2 -14829.865} C_VEL
LIN {X 0,Y 330.209,Z 580.998,A -85,B 0,C 180,E1 -14831.382,E2 -14831.382} C_VEL
LIN {X 0,Y 328.667,Z 591.267,A -85,B 0,C 180,E1 -14833.221,E2 -14833.221} C_VEL
LIN {X 0,Y 327.518,Z 599.781,A -85,B 0,C 180,E1 -14835.078,E2 -14835.078} C_VEL
LIN {X 0,Y 326.472,Z 607.904,A -85,B 0,C 180,E1 -14837.253,E2 -14837.253} C_VEL
LIN {X 0,Y 325.619,Z 614.44,A -85,B 0,C 180,E1 -14839.429,E2 -14839.429} C_VEL
LIN {X 0,Y 325.151,Z 620.236,A -85,B 0,C 180,E1 -14841.924,E2 -14841.924} C_VEL
LIN {X 0,Y 324.983,Z 624.053,A -85,B 0,C 180,E1 -14844.145,E2 -14844.145} C_VEL
LIN {X 0,Y 324.895,Z 626.63,A -85,B 0,C 180,E1 -14846.279,E2 -14846.279} C_VEL
LIN {X 0,Y 324.834,Z 628.331,A -85,B 0,C 180,E1 -14848.76,E2 -14848.76} C_VEL
LIN {X 0,Y 324.874,Z 628.677,A -85,B 0,C 180,E1 -14850,E2 -14850} C_VEL
LIN {X 0,Y 324.83,Z 628.365,A -85,B 0,C 180,E1 -14852.48,E2 -14852.48} C_VEL
LIN {X 0,Y 324.873,Z 626.718,A -85,B 0,C 180,E1 -14854.964,E2 -14854.964} C_VEL
LIN {X 0,Y 325.104,Z 623.707,A -85,B 0,C 180,E1 -14857.453,E2 -14857.453} C_VEL
LIN {X 0,Y 325.568,Z 619.25,A -85,B 0,C 180,E1 -14859.945,E2 -14859.945} C_VEL
LIN {X 0,Y 326.183,Z 614.848,A -85,B 0,C 180,E1 -14861.811,E2 -14861.811} C_VEL
LIN {X 0,Y 327.328,Z 608.494,A -85,B 0,C 180,E1 -14863.978,E2 -14863.978} C_VEL
LIN {X 0,Y 328.628,Z 600.606,A -85,B 0,C 180,E1 -14866.142,E2 -14866.142} C_VEL
LIN {X 0,Y 330.214,Z 592.383,A -85,B 0,C 180,E1 -14867.975,E2 -14867.975} C_VEL
LIN {X 0,Y 332.127,Z 582.496,A -85,B 0,C 180,E1 -14869.79,E2 -14869.79} C_VEL
LIN {X 0,Y 334.203,Z 571.523,A -85,B 0,C 180,E1 -14871.431,E2 -14871.431} C_VEL
LIN {X 0,Y 336.178,Z 559.801,A -85,B 0,C 180,E1 -14872.859,E2 -14872.859} C_VEL
LIN {X 0,Y 337.993,Z 547.287,A -85,B 0,C 180,E1 -14874.083,E2 -14874.083} C_VEL
LIN {X 0,Y 339.731,Z 533.936,A -85,B 0,C 180,E1 -14875.093,E2 -14875.093} C_VEL
LIN {X 0,Y 341.235,Z 520.049,A -85,B 0,C 180,E1 -14875.873,E2 -14875.873} C_VEL
LIN {X 0,Y 342.353,Z 505.516,A -85,B 0,C 180,E1 -14876.437,E2 -14876.437} C_VEL
LIN {X 0,Y 343.094,Z 483.528,A -85,B 0,C 180,E1 -14876.95,E2 -14876.95} C_VEL
LIN {X 0,Y 345.115,Z 409.498,A -85,B 0,C 180,E1 -14878.5,E2 -14878.5} C_VEL
LIN {X 0,Y 340.105,Z 383.141,A -85,B 0,C 180,E1 -14879.633,E2 -14879.633} C_VEL
LIN {X 0,Y 336.709,Z 375.032,A -85,B 0,C 180,E1 -14880.188,E2 -14880.188} C_VEL
LIN {X 0,Y 332.057,Z 364.769,A -85,B 0,C 180,E1 -14880.966,E2 -14880.966} C_VEL
LIN {X 0,Y 329.167,Z 352.777,A -85,B 0,C 180,E1 -14884.457,E2 -14884.457} C_VEL
LIN {X 0,Y 326.608,Z 343.425,A -85,B 0,C 180,E1 -14887.406,E2 -14887.406} C_VEL
LIN {X 0,Y 326.578,Z 343.428,A -85,B 0,C 180,E1 -14891.132,E2 -14891.132} C_VEL
LIN {X 0,Y 326.528,Z 343.436,A -85,B 0,C 180,E1 -14894.743,E2 -14894.743} C_VEL
LIN {X 0,Y 326.577,Z 343.426,A -85,B 0,C 180,E1 -14898.155,E2 -14898.155} C_VEL
LIN {X 0,Y 326.626,Z 343.42,A -85,B 0,C 180,E1 -14901.392,E2 -14901.392} C_VEL
LIN {X 0,Y 326.622,Z 343.425,A -85,B 0,C 180,E1 -14904.851,E2 -14904.851} C_VEL
LIN {X 0,Y 326.609,Z 343.422,A -85,B 0,C 180,E1 -14907.456,E2 -14907.456} C_VEL
LIN {X 0,Y 326.619,Z 343.42,A -85,B 0,C 180,E1 -14910.337,E2 -14910.337} C_VEL
LIN {X 0,Y 326.62,Z 343.42,A -85,B 0,C 180,E1 -14913.137,E2 -14913.137} C_VEL
LIN {X 0,Y 326.643,Z 343.422,A -85,B 0,C 180,E1 -14915.871,E2 -14915.871} C_VEL
LIN {X 0,Y 326.663,Z 343.42,A -85,B 0,C 180,E1 -14919.865,E2 -14919.865} C_VEL
LIN {X 0,Y 326.702,Z 343.406,A -85,B 0,C 180,E1 -14922.473,E2 -14922.473} C_VEL
LIN {X 0,Y 326.762,Z 343.397,A -85,B 0,C 180,E1 -14926.315,E2 -14926.315} C_VEL
LIN {X 0,Y 326.807,Z 343.399,A -85,B 0,C 180,E1 -14930.094,E2 -14930.094} C_VEL
LIN {X 0,Y 326.947,Z 343.384,A -85,B 0,C 180,E1 -14933.83,E2 -14933.83} C_VEL
LIN {X 0,Y 327.014,Z 343.366,A -85,B 0,C 180,E1 -14937.537,E2 -14937.537} C_VEL
LIN {X 0,Y 327.034,Z 343.365,A -85,B 0,C 180,E1 -14941.232,E2 -14941.232} C_VEL
LIN {X 0,Y 327.037,Z 343.365,A -85,B 0,C 180,E1 -14942.464,E2 -14942.464} C_VEL
LIN {X 0,Y 326.926,Z 343.374,A -85,B 0,C 180,E1 -14946.448,E2 -14946.448} C_VEL
LIN {X 0,Y 326.787,Z 343.403,A -85,B 0,C 180,E1 -14949.907,E2 -14949.907} C_VEL
LIN {X 0,Y 326.746,Z 343.409,A -85,B 0,C 180,E1 -14953.686,E2 -14953.686} C_VEL
LIN {X 0,Y 326.63,Z 343.418,A -85,B 0,C 180,E1 -14957.532,E2 -14957.532} C_VEL
LIN {X 0,Y 326.605,Z 343.419,A -85,B 0,C 180,E1 -14961.458,E2 -14961.458} C_VEL
LIN {X 0,Y 326.603,Z 343.421,A -85,B 0,C 180,E1 -14965.492,E2 -14965.492} C_VEL
LIN {X 0,Y 326.592,Z 343.42,A -85,B 0,C 180,E1 -14968.257,E2 -14968.257} C_VEL
LIN {X 0,Y 326.57,Z 343.404,A -85,B 0,C 180,E1 -14971.098,E2 -14971.098} C_VEL
LIN {X 0,Y 326.609,Z 343.425,A -85,B 0,C 180,E1 -14974.02,E2 -14974.02} C_VEL
LIN {X 0,Y 326.624,Z 343.404,A -85,B 0,C 180,E1 -14977.237,E2 -14977.237} C_VEL
LIN {X 0,Y 326.546,Z 343.433,A -85,B 0,C 180,E1 -14981.124,E2 -14981.124} C_VEL
LIN {X 0,Y 326.562,Z 343.434,A -85,B 0,C 180,E1 -14983.526,E2 -14983.526} C_VEL
LIN {X 0,Y 326.575,Z 343.429,A -85,B 0,C 180,E1 -14987.029,E2 -14987.029} C_VEL
LIN {X 0,Y 326.614,Z 343.429,A -85,B 0,C 180,E1 -14991.39,E2 -14991.39} C_VEL
LIN {X 0,Y 326.635,Z 343.574,A -85,B 0,C 180,E1 -14991.651,E2 -14991.651} C_VEL
LIN {X 0,Y 328.206,Z 349.612,A -85,B 0,C 180,E1 -14993.664,E2 -14993.664} C_VEL
LIN {X 0,Y 337.188,Z 367.424,A -85,B 0,C 180,E1 -14995.114,E2 -14995.114} C_VEL
LIN {X 0,Y 345.043,Z 385.167,A -85,B 0,C 180,E1 -14996.354,E2 -14996.354} C_VEL
LIN {X 0,Y 345.713,Z 386.826,A -85,B 0,C 180,E1 -14996.46,E2 -14996.46} C_VEL
LIN {X 0,Y 342.945,Z 486.353,A -85,B 0,C 180,E1 -14998.581,E2 -14998.581} C_VEL
LIN {X 0,Y 341.983,Z 501.021,A -85,B 0,C 180,E1 -14999.132,E2 -14999.132} C_VEL
LIN {X 0,Y 340.572,Z 515.476,A -85,B 0,C 180,E1 -14999.93,E2 -14999.93} C_VEL
LIN {X 0,Y 339.202,Z 527.273,A -85,B 0,C 180,E1 -15000.803,E2 -15000.803} C_VEL
LIN {X 0,Y 337.58,Z 539.039,A -85,B 0,C 180,E1 -15001.899,E2 -15001.899} C_VEL
LIN {X 0,Y 335.671,Z 550.745,A -85,B 0,C 180,E1 -15003.246,E2 -15003.246} C_VEL
LIN {X 0,Y 333.777,Z 561.643,A -85,B 0,C 180,E1 -15004.795,E2 -15004.795} C_VEL
LIN {X 0,Y 331.842,Z 572.024,A -85,B 0,C 180,E1 -15006.603,E2 -15006.603} C_VEL
LIN {X 0,Y 330.108,Z 580.722,A -85,B 0,C 180,E1 -15008.454,E2 -15008.454} C_VEL
LIN {X 0,Y 328.466,Z 589.21,A -85,B 0,C 180,E1 -15010.688,E2 -15010.688} C_VEL
LIN {X 0,Y 327.362,Z 594.801,A -85,B 0,C 180,E1 -15012.509,E2 -15012.509} C_VEL
LIN {X 0,Y 326.542,Z 599.523,A -85,B 0,C 180,E1 -15014.393,E2 -15014.393} C_VEL
LIN {X 0,Y 325.661,Z 604.395,A -85,B 0,C 180,E1 -15016.903,E2 -15016.903} C_VEL
LIN {X 0,Y 325.203,Z 607.036,A -85,B 0,C 180,E1 -15018.784,E2 -15018.784} C_VEL
LIN {X 0,Y 324.946,Z 609.322,A -85,B 0,C 180,E1 -15021.292,E2 -15021.292} C_VEL
LIN {X 0,Y 324.945,Z 610.261,A -85,B 0,C 180,E1 -15023.792,E2 -15023.792} C_VEL
LIN {X 0,Y 324.898,Z 609.887,A -85,B 0,C 180,E1 -15026.279,E2 -15026.279} C_VEL
LIN {X 0,Y 324.902,Z 608.198,A -85,B 0,C 180,E1 -15028.76,E2 -15028.76} C_VEL
LIN {X 0,Y 325.143,Z 605.159,A -85,B 0,C 180,E1 -15031.239,E2 -15031.239} C_VEL
LIN {X 0,Y 325.624,Z 600.686,A -85,B 0,C 180,E1 -15033.712,E2 -15033.712} C_VEL
LIN {X 0,Y 326.378,Z 596.241,A -85,B 0,C 180,E1 -15035.561,E2 -15035.561} C_VEL
LIN {X 0,Y 327.169,Z 589.859,A -85,B 0,C 180,E1 -15037.716,E2 -15037.716} C_VEL
LIN {X 0,Y 328.299,Z 581.941,A -85,B 0,C 180,E1 -15039.861,E2 -15039.861} C_VEL
LIN {X 0,Y 329.475,Z 573.661,A -85,B 0,C 180,E1 -15041.692,E2 -15041.692} C_VEL
LIN {X 0,Y 331.139,Z 563.679,A -85,B 0,C 180,E1 -15043.501,E2 -15043.501} C_VEL
LIN {X 0,Y 332.667,Z 552.551,A -85,B 0,C 180,E1 -15045.155,E2 -15045.155} C_VEL
LIN {X 0,Y 334.105,Z 541.488,A -85,B 0,C 180,E1 -15046.498,E2 -15046.498} C_VEL
LIN {X 0,Y 335.571,Z 529.437,A -85,B 0,C 180,E1 -15047.679,E2 -15047.679} C_VEL
LIN {X 0,Y 336.879,Z 516.096,A -85,B 0,C 180,E1 -15048.709,E2 -15048.709} C_VEL
LIN {X 0,Y 338.007,Z 502.145,A -85,B 0,C 180,E1 -15049.511,E2 -15049.511} C_VEL
LIN {X 0,Y 338.789,Z 487.44,A -85,B 0,C 180,E1 -15050.095,E2 -15050.095} C_VEL
LIN {X 0,Y 339.548,Z 460.703,A -85,B 0,C 180,E1 -15050.7,E2 -15050.7} C_VEL
LIN {X 0,Y 341.364,Z 383.243,A -85,B 0,C 180,E1 -15052.322,E2 -15052.322} C_VEL
LIN {X 0,Y 340.13,Z 378.69,A -85,B 0,C 180,E1 -15052.526,E2 -15052.526} C_VEL
LIN {X 0,Y 337.105,Z 370.946,A -85,B 0,C 180,E1 -15052.953,E2 -15052.953} C_VEL
LIN {X 0,Y 335.042,Z 367.837,A -85,B 0,C 180,E1 -15053.199,E2 -15053.199} C_VEL
LIN {X 0,Y 325.907,Z 359.711,A -85,B 0,C 180,E1 -15054.193,E2 -15054.193} C_VEL
LIN {X 0,Y 323.987,Z 356.543,A -85,B 0,C 180,E1 -15054.446,E2 -15054.446} C_VEL
LIN {X 0,Y 320.734,Z 349.31,A -85,B 0,C 180,E1 -15054.96,E2 -15054.96} C_VEL
LIN {X 0,Y 319.55,Z 344.31,A -85,B 0,C 180,E1 -15056.535,E2 -15056.535} C_VEL
LIN {X 0,Y 319.555,Z 344.298,A -85,B 0,C 180,E1 -15060.387,E2 -15060.387} C_VEL
LIN {X 0,Y 319.579,Z 344.303,A -85,B 0,C 180,E1 -15063.353,E2 -15063.353} C_VEL
LIN {X 0,Y 319.557,Z 344.304,A -85,B 0,C 180,E1 -15066.428,E2 -15066.428} C_VEL
LIN {X 0,Y 319.531,Z 344.305,A -85,B 0,C 180,E1 -15069.662,E2 -15069.662} C_VEL
LIN {X 0,Y 319.521,Z 344.308,A -85,B 0,C 180,E1 -15073.46,E2 -15073.46} C_VEL
LIN {X 0,Y 319.553,Z 344.305,A -85,B 0,C 180,E1 -15077.016,E2 -15077.016} C_VEL
LIN {X 0,Y 319.548,Z 344.306,A -85,B 0,C 180,E1 -15080.37,E2 -15080.37} C_VEL
LIN {X 0,Y 319.582,Z 344.301,A -85,B 0,C 180,E1 -15084.457,E2 -15084.457} C_VEL
LIN {X 0,Y 319.527,Z 344.3,A -85,B 0,C 180,E1 -15088.137,E2 -15088.137} C_VEL
LIN {X 0,Y 319.546,Z 344.3,A -85,B 0,C 180,E1 -15091.613,E2 -15091.613} C_VEL
LIN {X 0,Y 319.543,Z 344.305,A -85,B 0,C 180,E1 -15095.298,E2 -15095.298} C_VEL
LIN {X 0,Y 319.566,Z 344.287,A -85,B 0,C 180,E1 -15098.045,E2 -15098.045} C_VEL
LIN {X 0,Y 319.589,Z 344.289,A -85,B 0,C 180,E1 -15102.069,E2 -15102.069} C_VEL
LIN {X 0,Y 319.712,Z 344.28,A -85,B 0,C 180,E1 -15106.006,E2 -15106.006} C_VEL
LIN {X 0,Y 319.738,Z 344.251,A -85,B 0,C 180,E1 -15109.872,E2 -15109.872} C_VEL
LIN {X 0,Y 319.904,Z 344.26,A -85,B 0,C 180,E1 -15113.693,E2 -15113.693} C_VEL
LIN {X 0,Y 319.98,Z 344.248,A -85,B 0,C 180,E1 -15117.482,E2 -15117.482} C_VEL
LIN {X 0,Y 320.016,Z 344.238,A -85,B 0,C 180,E1 -15121.258,E2 -15121.258} C_VEL
LIN {X 0,Y 319.723,Z 344.278,A -85,B 0,C 180,E1 -15125.044,E2 -15125.044} C_VEL
LIN {X 0,Y 319.856,Z 344.266,A -85,B 0,C 180,E1 -15127.575,E2 -15127.575} C_VEL
LIN {X 0,Y 319.718,Z 344.282,A -85,B 0,C 180,E1 -15131.41,E2 -15131.41} C_VEL
LIN {X 0,Y 319.702,Z 344.282,A -85,B 0,C 180,E1 -15135.295,E2 -15135.295} C_VEL
LIN {X 0,Y 319.676,Z 344.286,A -85,B 0,C 180,E1 -15139.255,E2 -15139.255} C_VEL
LIN {X 0,Y 319.57,Z 344.301,A -85,B 0,C 180,E1 -15143.319,E2 -15143.319} C_VEL
LIN {X 0,Y 319.59,Z 344.299,A -85,B 0,C 180,E1 -15146.092,E2 -15146.092} C_VEL
LIN {X 0,Y 319.565,Z 344.302,A -85,B 0,C 180,E1 -15148.936,E2 -15148.936} C_VEL
LIN {X 0,Y 319.527,Z 344.309,A -85,B 0,C 180,E1 -15151.862,E2 -15151.862} C_VEL
LIN {X 0,Y 319.582,Z 344.302,A -85,B 0,C 180,E1 -15155.543,E2 -15155.543} C_VEL
LIN {X 0,Y 319.575,Z 344.302,A -85,B 0,C 180,E1 -15158.007,E2 -15158.007} C_VEL
LIN {X 0,Y 319.527,Z 344.312,A -85,B 0,C 180,E1 -15161.597,E2 -15161.597} C_VEL
LIN {X 0,Y 319.489,Z 344.315,A -85,B 0,C 180,E1 -15165.257,E2 -15165.257} C_VEL
LIN {X 0,Y 319.529,Z 344.308,A -85,B 0,C 180,E1 -15168.712,E2 -15168.712} C_VEL
LIN {X 0,Y 319.578,Z 344.308,A -85,B 0,C 180,E1 -15172.344,E2 -15172.344} C_VEL
LIN {X 0,Y 319.607,Z 344.381,A -85,B 0,C 180,E1 -15174.649,E2 -15174.649} C_VEL
LIN {X 0,Y 322.544,Z 356.732,A -85,B 0,C 180,E1 -15178.188,E2 -15178.188} C_VEL
LIN {X 0,Y 324.376,Z 364.921,A -85,B 0,C 180,E1 -15180.424,E2 -15180.424} C_VEL
LIN {X 0,Y 329.333,Z 378.093,A -85,B 0,C 180,E1 -15181.193,E2 -15181.193} C_VEL
LIN {X 0,Y 333.545,Z 403.564,A -85,B 0,C 180,E1 -15182.152,E2 -15182.152} C_VEL
LIN {X 0,Y 334.497,Z 410.073,A -85,B 0,C 180,E1 -15182.382,E2 -15182.382} C_VEL
LIN {X 0,Y 332.136,Z 502.725,A -85,B 0,C 180,E1 -15184.376,E2 -15184.376} C_VEL
LIN {X 0,Y 331.163,Z 517.565,A -85,B 0,C 180,E1 -15184.926,E2 -15184.926} C_VEL
LIN {X 0,Y 329.884,Z 531.648,A -85,B 0,C 180,E1 -15185.704,E2 -15185.704} C_VEL
LIN {X 0,Y 328.356,Z 545.432,A -85,B 0,C 180,E1 -15186.74,E2 -15186.74} C_VEL
LIN {X 0,Y 326.871,Z 557.628,A -85,B 0,C 180,E1 -15187.924,E2 -15187.924} C_VEL
LIN {X 0,Y 325.041,Z 570.125,A -85,B 0,C 180,E1 -15189.43,E2 -15189.43} C_VEL
LIN {X 0,Y 323.421,Z 580.52,A -85,B 0,C 180,E1 -15190.977,E2 -15190.977} C_VEL
LIN {X 0,Y 321.812,Z 590.854,A -85,B 0,C 180,E1 -15192.853,E2 -15192.853} C_VEL
LIN {X 0,Y 320.572,Z 599.403,A -85,B 0,C 180,E1 -15194.747,E2 -15194.747} C_VEL
LIN {X 0,Y 319.624,Z 606.518,A -85,B 0,C 180,E1 -15196.651,E2 -15196.651} C_VEL
LIN {X 0,Y 318.778,Z 612.395,A -85,B 0,C 180,E1 -15198.555,E2 -15198.555} C_VEL
LIN {X 0,Y 318.275,Z 617.244,A -85,B 0,C 180,E1 -15200.467,E2 -15200.467} C_VEL
LIN {X 0,Y 317.968,Z 622.254,A -85,B 0,C 180,E1 -15203.018,E2 -15203.018} C_VEL
LIN {X 0,Y 317.814,Z 625.011,A -85,B 0,C 180,E1 -15204.925,E2 -15204.925} C_VEL
LIN {X 0,Y 317.762,Z 627.421,A -85,B 0,C 180,E1 -15207.465,E2 -15207.465} C_VEL
LIN {X 0,Y 317.781,Z 628.47,A -85,B 0,C 180,E1 -15210,E2 -15210} C_VEL
LIN {X 0,Y 317.751,Z 628.18,A -85,B 0,C 180,E1 -15212.535,E2 -15212.535} C_VEL
LIN {X 0,Y 317.789,Z 626.555,A -85,B 0,C 180,E1 -15215.075,E2 -15215.075} C_VEL
LIN {X 0,Y 318.024,Z 623.566,A -85,B 0,C 180,E1 -15217.62,E2 -15217.62} C_VEL
LIN {X 0,Y 318.533,Z 619.133,A -85,B 0,C 180,E1 -15220.167,E2 -15220.167} C_VEL
LIN {X 0,Y 319.534,Z 613.129,A -85,B 0,C 180,E1 -15222.706,E2 -15222.706} C_VEL
LIN {X 0,Y 320.737,Z 606.388,A -85,B 0,C 180,E1 -15224.92,E2 -15224.92} C_VEL
LIN {X 0,Y 322.293,Z 598.023,A -85,B 0,C 180,E1 -15227.121,E2 -15227.121} C_VEL
LIN {X 0,Y 324.052,Z 589.326,A -85,B 0,C 180,E1 -15228.985,E2 -15228.985} C_VEL
LIN {X 0,Y 326.173,Z 578.806,A -85,B 0,C 180,E1 -15230.826,E2 -15230.826} C_VEL
LIN {X 0,Y 328.42,Z 567.049,A -85,B 0,C 180,E1 -15232.49,E2 -15232.49} C_VEL
LIN {X 0,Y 330.374,Z 555.276,A -85,B 0,C 180,E1 -15233.84,E2 -15233.84} C_VEL
LIN {X 0,Y 332.276,Z 542.299,A -85,B 0,C 180,E1 -15235.026,E2 -15235.026} C_VEL
LIN {X 0,Y 334.011,Z 528.722,A -85,B 0,C 180,E1 -15235.972,E2 -15235.972} C_VEL
LIN {X 0,Y 335.461,Z 514.406,A -85,B 0,C 180,E1 -15236.688,E2 -15236.688} C_VEL
LIN {X 0,Y 336.337,Z 500.454,A -85,B 0,C 180,E1 -15237.158,E2 -15237.158} C_VEL
LIN {X 0,Y 339.004,Z 411.067,A -85,B 0,C 180,E1 -15239.069,E2 -15239.069} C_VEL
LIN {X 0,Y 334.473,Z 386.403,A -85,B 0,C 180,E1 -15240.145,E2 -15240.145} C_VEL
LIN {X 0,Y 332.014,Z 380.08,A -85,B 0,C 180,E1 -15240.569,E2 -15240.569} C_VEL
LIN {X 0,Y 324.774,Z 364.448,A -85,B 0,C 180,E1 -15241.828,E2 -15241.828} C_VEL
LIN {X 0,Y 322.276,Z 354.225,A -85,B 0,C 180,E1 -15244.904,E2 -15244.904} C_VEL
LIN {X 0,Y 319.552,Z 344.295,A -85,B 0,C 180,E1 -15248.111,E2 -15248.111} C_VEL
LIN {X 0,Y 319.526,Z 344.306,A -85,B 0,C 180,E1 -15251.597,E2 -15251.597} C_VEL
LIN {X 0,Y 319.489,Z 344.31,A -85,B 0,C 180,E1 -15255.258,E2 -15255.258} C_VEL
LIN {X 0,Y 319.53,Z 344.305,A -85,B 0,C 180,E1 -15258.712,E2 -15258.712} C_VEL
LIN {X 0,Y 319.58,Z 344.303,A -85,B 0,C 180,E1 -15262.344,E2 -15262.344} C_VEL
LIN {X 0,Y 319.562,Z 344.303,A -85,B 0,C 180,E1 -15265.124,E2 -15265.124} C_VEL
LIN {X 0,Y 319.526,Z 344.308,A -85,B 0,C 180,E1 -15268.138,E2 -15268.138} C_VEL
LIN {X 0,Y 319.59,Z 344.299,A -85,B 0,C 180,E1 -15271.598,E2 -15271.598} C_VEL
LIN {X 0,Y 319.583,Z 344.299,A -85,B 0,C 180,E1 -15275.302,E2 -15275.302} C_VEL
LIN {X 0,Y 319.606,Z 344.296,A -85,B 0,C 180,E1 -15279.401,E2 -15279.401} C_VEL
LIN {X 0,Y 319.661,Z 344.283,A -85,B 0,C 180,E1 -15282.074,E2 -15282.074} C_VEL
LIN {X 0,Y 319.735,Z 344.275,A -85,B 0,C 180,E1 -15286.008,E2 -15286.008} C_VEL
LIN {X 0,Y 319.754,Z 344.28,A -85,B 0,C 180,E1 -15289.873,E2 -15289.873} C_VEL
LIN {X 0,Y 319.904,Z 344.26,A -85,B 0,C 180,E1 -15293.694,E2 -15293.694} C_VEL
LIN {X 0,Y 319.96,Z 344.244,A -85,B 0,C 180,E1 -15297.483,E2 -15297.483} C_VEL
LIN {X 0,Y 320.004,Z 344.24,A -85,B 0,C 180,E1 -15301.259,E2 -15301.259} C_VEL
LIN {X 0,Y 319.719,Z 344.284,A -85,B 0,C 180,E1 -15303.782,E2 -15303.782} C_VEL
LIN {X 0,Y 319.892,Z 344.25,A -85,B 0,C 180,E1 -15306.428,E2 -15306.428} C_VEL
LIN {X 0,Y 319.739,Z 344.279,A -85,B 0,C 180,E1 -15310.128,E2 -15310.128} C_VEL
LIN {X 0,Y 319.713,Z 344.286,A -85,B 0,C 180,E1 -15313.994,E2 -15313.994} C_VEL
LIN {X 0,Y 319.581,Z 344.301,A -85,B 0,C 180,E1 -15317.932,E2 -15317.932} C_VEL
LIN {X 0,Y 319.563,Z 344.302,A -85,B 0,C 180,E1 -15321.955,E2 -15321.955} C_VEL
LIN {X 0,Y 319.552,Z 344.305,A -85,B 0,C 180,E1 -15326.096,E2 -15326.096} C_VEL
LIN {X 0,Y 319.526,Z 344.289,A -85,B 0,C 180,E1 -15328.94,E2 -15328.94} C_VEL
LIN {X 0,Y 319.523,Z 344.291,A -85,B 0,C 180,E1 -15331.863,E2 -15331.863} C_VEL
LIN {X 0,Y 319.581,Z 344.284,A -85,B 0,C 180,E1 -15335.542,E2 -15335.542} C_VEL
LIN {X 0,Y 319.531,Z 344.306,A -85,B 0,C 180,E1 -15339.662,E2 -15339.662} C_VEL
LIN {X 0,Y 319.521,Z 344.311,A -85,B 0,C 180,E1 -15343.46,E2 -15343.46} C_VEL
LIN {X 0,Y 319.553,Z 344.303,A -85,B 0,C 180,E1 -15347.016,E2 -15347.016} C_VEL
LIN {X 0,Y 319.58,Z 344.413,A -85,B 0,C 180,E1 -15350.935,E2 -15350.935} C_VEL
LIN {X 0,Y 321.106,Z 350.075,A -85,B 0,C 180,E1 -15352.828,E2 -15352.828} C_VEL
LIN {X 0,Y 330.479,Z 368.183,A -85,B 0,C 180,E1 -15354.399,E2 -15354.399} C_VEL
LIN {X 0,Y 339.265,Z 387.902,A -85,B 0,C 180,E1 -15355.834,E2 -15355.834} C_VEL
LIN {X 0,Y 339.59,Z 389.483,A -85,B 0,C 180,E1 -15355.906,E2 -15355.906} C_VEL
LIN {X 0,Y 336.776,Z 485.775,A -85,B 0,C 180,E1 -15357.981,E2 -15357.981} C_VEL
LIN {X 0,Y 335.875,Z 499.878,A -85,B 0,C 180,E1 -15358.502,E2 -15358.502} C_VEL
LIN {X 0,Y 334.454,Z 514.162,A -85,B 0,C 180,E1 -15359.277,E2 -15359.277} C_VEL
LIN {X 0,Y 332.87,Z 527.325,A -85,B 0,C 180,E1 -15360.25,E2 -15360.25} C_VEL
LIN {X 0,Y 331.028,Z 540.083,A -85,B 0,C 180,E1 -15361.465,E2 -15361.465} C_VEL
LIN {X 0,Y 329.051,Z 551.639,A -85,B 0,C 180,E1 -15362.836,E2 -15362.836} C_VEL
LIN {X 0,Y 327.261,Z 561.436,A -85,B 0,C 180,E1 -15364.257,E2 -15364.257} C_VEL
LIN {X 0,Y 325.258,Z 571.885,A -85,B 0,C 180,E1 -15366.1,E2 -15366.1} C_VEL
LIN {X 0,Y 323.391,Z 580.64,A -85,B 0,C 180,E1 -15367.983,E2 -15367.983} C_VEL
LIN {X 0,Y 321.928,Z 587.735,A -85,B 0,C 180,E1 -15369.841,E2 -15369.841} C_VEL
LIN {X 0,Y 320.483,Z 594.814,A -85,B 0,C 180,E1 -15372.121,E2 -15372.121} C_VEL
LIN {X 0,Y 319.596,Z 599.576,A -85,B 0,C 180,E1 -15374.045,E2 -15374.045} C_VEL
LIN {X 0,Y 318.669,Z 604.486,A -85,B 0,C 180,E1 -15376.61,E2 -15376.61} C_VEL
LIN {X 0,Y 318.179,Z 607.163,A -85,B 0,C 180,E1 -15378.533,E2 -15378.533} C_VEL
LIN {X 0,Y 317.861,Z 609.483,A -85,B 0,C 180,E1 -15381.096,E2 -15381.096} C_VEL
LIN {X 0,Y 317.85,Z 610.455,A -85,B 0,C 180,E1 -15383.653,E2 -15383.653} C_VEL
LIN {X 0,Y 317.805,Z 610.113,A -85,B 0,C 180,E1 -15386.196,E2 -15386.196} C_VEL
LIN {X 0,Y 317.81,Z 608.458,A -85,B 0,C 180,E1 -15388.733,E2 -15388.733} C_VEL
LIN {X 0,Y 318.05,Z 605.453,A -85,B 0,C 180,E1 -15391.266,E2 -15391.266} C_VEL
LIN {X 0,Y 318.547,Z 601.02,A -85,B 0,C 180,E1 -15393.795,E2 -15393.795} C_VEL
LIN {X 0,Y 319.325,Z 596.61,A -85,B 0,C 180,E1 -15395.684,E2 -15395.684} C_VEL
LIN {X 0,Y 320.165,Z 590.269,A -85,B 0,C 180,E1 -15397.886,E2 -15397.886} C_VEL
LIN {X 0,Y 321.329,Z 582.397,A -85,B 0,C 180,E1 -15400.077,E2 -15400.077} C_VEL
LIN {X 0,Y 322.278,Z 575.645,A -85,B 0,C 180,E1 -15401.637,E2 -15401.637} C_VEL
LIN {X 0,Y 324.027,Z 566.01,A -85,B 0,C 180,E1 -15403.483,E2 -15403.483} C_VEL
LIN {X 0,Y 325.607,Z 555.348,A -85,B 0,C 180,E1 -15405.172,E2 -15405.172} C_VEL
LIN {X 0,Y 327.172,Z 543.548,A -85,B 0,C 180,E1 -15406.697,E2 -15406.697} C_VEL
LIN {X 0,Y 328.675,Z 531.942,A -85,B 0,C 180,E1 -15407.901,E2 -15407.901} C_VEL
LIN {X 0,Y 330.103,Z 518.317,A -85,B 0,C 180,E1 -15409.027,E2 -15409.027} C_VEL
LIN {X 0,Y 331.328,Z 504.356,A -85,B 0,C 180,E1 -15409.88,E2 -15409.88} C_VEL
LIN {X 0,Y 332.147,Z 490.645,A -85,B 0,C 180,E1 -15410.475,E2 -15410.475} C_VEL
LIN {X 0,Y 332.699,Z 475.288,A -85,B 0,C 180,E1 -15410.884,E2 -15410.884} C_VEL
LIN {X 0,Y 334.947,Z 384.387,A -85,B 0,C 180,E1 -15412.819,E2 -15412.819} C_VEL
LIN {X 0,Y 332.016,Z 375.963,A -85,B 0,C 180,E1 -15413.265,E2 -15413.265} C_VEL
LIN {X 0,Y 323.987,Z 356.543,A -85,B 0,C 180,E1 -15414.446,E2 -15414.446} C_VEL
LIN {X 0,Y 322.009,Z 353.428,A -85,B 0,C 180,E1 -15414.733,E2 -15414.733} C_VEL
LIN {X 0,Y 319.386,Z 351.143,A -85,B 0,C 180,E1 -15415.124,E2 -15415.124} C_VEL
LIN {X 0,Y 315.027,Z 348.327,A -85,B 0,C 180,E1 -15415.957,E2 -15415.957} C_VEL
LIN {X 0,Y 312.943,Z 346.374,A -85,B 0,C 180,E1 -15416.664,E2 -15416.664} C_VEL
LIN {X 0,Y 312.564,Z 345.404,A -85,B 0,C 180,E1 -15416.987,E2 -15416.987} C_VEL
LIN {X 0,Y 312.492,Z 345.189,A -85,B 0,C 180,E1 -15417.455,E2 -15417.455} C_VEL
LIN {X 0,Y 312.5,Z 345.183,A -85,B 0,C 180,E1 -15421.283,E2 -15421.283} C_VEL
LIN {X 0,Y 312.508,Z 345.183,A -85,B 0,C 180,E1 -15424.21,E2 -15424.21} C_VEL
LIN {X 0,Y 312.512,Z 345.182,A -85,B 0,C 180,E1 -15427.387,E2 -15427.387} C_VEL
LIN {X 0,Y 312.443,Z 345.193,A -85,B 0,C 180,E1 -15430.717,E2 -15430.717} C_VEL
LIN {X 0,Y 312.452,Z 345.19,A -85,B 0,C 180,E1 -15434.21,E2 -15434.21} C_VEL
LIN {X 0,Y 312.456,Z 345.187,A -85,B 0,C 180,E1 -15437.925,E2 -15437.925} C_VEL
LIN {X 0,Y 312.479,Z 345.184,A -85,B 0,C 180,E1 -15441.924,E2 -15441.924} C_VEL
LIN {X 0,Y 312.534,Z 345.177,A -85,B 0,C 180,E1 -15444.22,E2 -15444.22} C_VEL
LIN {X 0,Y 312.504,Z 345.172,A -85,B 0,C 180,E1 -15447.333,E2 -15447.333} C_VEL
LIN {X 0,Y 312.486,Z 345.18,A -85,B 0,C 180,E1 -15451.299,E2 -15451.299} C_VEL
LIN {X 0,Y 312.524,Z 345.182,A -85,B 0,C 180,E1 -15454.705,E2 -15454.705} C_VEL
LIN {X 0,Y 312.542,Z 345.17,A -85,B 0,C 180,E1 -15457.525,E2 -15457.525} C_VEL
LIN {X 0,Y 312.553,Z 345.163,A -85,B 0,C 180,E1 -15461.651,E2 -15461.651} C_VEL
LIN {X 0,Y 312.654,Z 345.162,A -85,B 0,C 180,E1 -15465.684,E2 -15465.684} C_VEL
LIN {X 0,Y 312.688,Z 345.127,A -85,B 0,C 180,E1 -15469.641,E2 -15469.641} C_VEL
LIN {X 0,Y 312.799,Z 345.141,A -85,B 0,C 180,E1 -15472.252,E2 -15472.252} C_VEL
LIN {X 0,Y 312.698,Z 345.156,A -85,B 0,C 180,E1 -15474.842,E2 -15474.842} C_VEL
LIN {X 0,Y 312.926,Z 345.126,A -85,B 0,C 180,E1 -15477.425,E2 -15477.425} C_VEL
LIN {X 0,Y 312.983,Z 345.114,A -85,B 0,C 180,E1 -15481.286,E2 -15481.286} C_VEL
LIN {X 0,Y 312.845,Z 345.139,A -85,B 0,C 180,E1 -15486.449,E2 -15486.449} C_VEL
LIN {X 0,Y 312.753,Z 345.149,A -85,B 0,C 180,E1 -15489.05,E2 -15489.05} C_VEL
LIN {X 0,Y 312.637,Z 345.164,A -85,B 0,C 180,E1 -15492.991,E2 -15492.991} C_VEL
LIN {X 0,Y 312.641,Z 345.164,A -85,B 0,C 180,E1 -15495.649,E2 -15495.649} C_VEL
LIN {X 0,Y 312.632,Z 345.163,A -85,B 0,C 180,E1 -15499.236,E2 -15499.236} C_VEL
LIN {X 0,Y 312.547,Z 345.175,A -85,B 0,C 180,E1 -15502.788,E2 -15502.788} C_VEL
LIN {X 0,Y 312.522,Z 345.18,A -85,B 0,C 180,E1 -15506.728,E2 -15506.728} C_VEL
LIN {X 0,Y 312.508,Z 345.182,A -85,B 0,C 180,E1 -15509.654,E2 -15509.654} C_VEL
LIN {X 0,Y 312.521,Z 345.185,A -85,B 0,C 180,E1 -15513.689,E2 -15513.689} C_VEL
LIN {X 0,Y 312.539,Z 345.184,A -85,B 0,C 180,E1 -15517.383,E2 -15517.383} C_VEL
LIN {X 0,Y 312.491,Z 345.186,A -85,B 0,C 180,E1 -15520.709,E2 -15520.709} C_VEL
LIN {X 0,Y 312.452,Z 345.191,A -85,B 0,C 180,E1 -15524.209,E2 -15524.209} C_VEL
LIN {X 0,Y 312.485,Z 345.184,A -85,B 0,C 180,E1 -15527.918,E2 -15527.918} C_VEL
LIN {X 0,Y 312.535,Z 345.183,A -85,B 0,C 180,E1 -15531.91,E2 -15531.91} C_VEL
LIN {X 0,Y 312.536,Z 345.314,A -85,B 0,C 180,E1 -15534.112,E2 -15534.112} C_VEL
LIN {X 0,Y 315.131,Z 355.92,A -85,B 0,C 180,E1 -15537.26,E2 -15537.26} C_VEL
LIN {X 0,Y 317.12,Z 364.674,A -85,B 0,C 180,E1 -15539.735,E2 -15539.735} C_VEL
LIN {X 0,Y 323.188,Z 380.224,A -85,B 0,C 180,E1 -15540.699,E2 -15540.699} C_VEL
LIN {X 0,Y 328.035,Z 409.944,A -85,B 0,C 180,E1 -15541.842,E2 -15541.842} C_VEL
LIN {X 0,Y 325.667,Z 502.336,A -85,B 0,C 180,E1 -15543.872,E2 -15543.872} C_VEL
LIN {X 0,Y 324.735,Z 516.49,A -85,B 0,C 180,E1 -15544.395,E2 -15544.395} C_VEL
LIN {X 0,Y 323.409,Z 530.799,A -85,B 0,C 180,E1 -15545.185,E2 -15545.185} C_VEL
LIN {X 0,Y 321.889,Z 544.011,A -85,B 0,C 180,E1 -15546.176,E2 -15546.176} C_VEL
LIN {X 0,Y 320.426,Z 555.849,A -85,B 0,C 180,E1 -15547.318,E2 -15547.318} C_VEL
LIN {X 0,Y 318.751,Z 567.222,A -85,B 0,C 180,E1 -15548.666,E2 -15548.666} C_VEL
LIN {X 0,Y 316.987,Z 578.071,A -85,B 0,C 180,E1 -15550.238,E2 -15550.238} C_VEL
LIN {X 0,Y 315.247,Z 588.806,A -85,B 0,C 180,E1 -15552.149,E2 -15552.149} C_VEL
LIN {X 0,Y 313.826,Z 597.663,A -85,B 0,C 180,E1 -15554.078,E2 -15554.078} C_VEL
LIN {X 0,Y 312.797,Z 605.027,A -85,B 0,C 180,E1 -15556.023,E2 -15556.023} C_VEL
LIN {X 0,Y 311.776,Z 612.064,A -85,B 0,C 180,E1 -15558.295,E2 -15558.295} C_VEL
LIN {X 0,Y 311.122,Z 618.381,A -85,B 0,C 180,E1 -15560.902,E2 -15560.902} C_VEL
LIN {X 0,Y 310.826,Z 623.013,A -85,B 0,C 180,E1 -15563.509,E2 -15563.509} C_VEL
LIN {X 0,Y 310.715,Z 626.149,A -85,B 0,C 180,E1 -15566.109,E2 -15566.109} C_VEL
LIN {X 0,Y 310.66,Z 627.895,A -85,B 0,C 180,E1 -15568.704,E2 -15568.704} C_VEL
LIN {X 0,Y 310.691,Z 628.263,A -85,B 0,C 180,E1 -15570,E2 -15570} C_VEL
LIN {X 0,Y 310.674,Z 627.995,A -85,B 0,C 180,E1 -15572.593,E2 -15572.593} C_VEL
LIN {X 0,Y 310.695,Z 626.392,A -85,B 0,C 180,E1 -15575.191,E2 -15575.191} C_VEL
LIN {X 0,Y 310.972,Z 623.427,A -85,B 0,C 180,E1 -15577.793,E2 -15577.793} C_VEL
LIN {X 0,Y 311.515,Z 619.018,A -85,B 0,C 180,E1 -15580.398,E2 -15580.398} C_VEL
LIN {X 0,Y 312.225,Z 614.669,A -85,B 0,C 180,E1 -15582.348,E2 -15582.348} C_VEL
LIN {X 0,Y 313.421,Z 608.371,A -85,B 0,C 180,E1 -15584.612,E2 -15584.612} C_VEL
LIN {X 0,Y 314.939,Z 600.549,A -85,B 0,C 180,E1 -15586.864,E2 -15586.864} C_VEL
LIN {X 0,Y 316.69,Z 592.399,A -85,B 0,C 180,E1 -15588.771,E2 -15588.771} C_VEL
LIN {X 0,Y 318.736,Z 582.596,A -85,B 0,C 180,E1 -15590.658,E2 -15590.658} C_VEL
LIN {X 0,Y 321.016,Z 571.726,A -85,B 0,C 180,E1 -15592.358,E2 -15592.358} C_VEL
LIN {X 0,Y 323.249,Z 559.537,A -85,B 0,C 180,E1 -15593.908,E2 -15593.908} C_VEL
LIN {X 0,Y 325.383,Z 546.123,A -85,B 0,C 180,E1 -15595.251,E2 -15595.251} C_VEL
LIN {X 0,Y 327.092,Z 533.698,A -85,B 0,C 180,E1 -15596.22,E2 -15596.22} C_VEL
LIN {X 0,Y 328.753,Z 519.864,A -85,B 0,C 180,E1 -15597.019,E2 -15597.019} C_VEL
LIN {X 0,Y 329.912,Z 505.447,A -85,B 0,C 180,E1 -15597.603,E2 -15597.603} C_VEL
LIN {X 0,Y 330.694,Z 485.524,A -85,B 0,C 180,E1 -15598.088,E2 -15598.088} C_VEL
LIN {X 0,Y 332.86,Z 411.41,A -85,B 0,C 180,E1 -15599.696,E2 -15599.696} C_VEL
LIN {X 0,Y 328.422,Z 387.797,A -85,B 0,C 180,E1 -15600.772,E2 -15600.772} C_VEL
LIN {X 0,Y 321.262,Z 372.076,A -85,B 0,C 180,E1 -15602.008,E2 -15602.008} C_VEL
LIN {X 0,Y 317.527,Z 364.3,A -85,B 0,C 180,E1 -15602.684,E2 -15602.684} C_VEL
LIN {X 0,Y 314.808,Z 353.386,A -85,B 0,C 180,E1 -15606.105,E2 -15606.105} C_VEL
LIN {X 0,Y 312.514,Z 345.17,A -85,B 0,C 180,E1 -15608.897,E2 -15608.897} C_VEL
LIN {X 0,Y 312.491,Z 345.188,A -85,B 0,C 180,E1 -15612.432,E2 -15612.432} C_VEL
LIN {X 0,Y 312.459,Z 345.185,A -85,B 0,C 180,E1 -15616.035,E2 -15616.035} C_VEL
LIN {X 0,Y 312.505,Z 345.182,A -85,B 0,C 180,E1 -15619.875,E2 -15619.875} C_VEL
LIN {X 0,Y 312.539,Z 345.177,A -85,B 0,C 180,E1 -15622.617,E2 -15622.617} C_VEL
LIN {X 0,Y 312.521,Z 345.177,A -85,B 0,C 180,E1 -15626.312,E2 -15626.312} C_VEL
LIN {X 0,Y 312.502,Z 345.178,A -85,B 0,C 180,E1 -15630.346,E2 -15630.346} C_VEL
LIN {X 0,Y 312.535,Z 345.172,A -85,B 0,C 180,E1 -15634.091,E2 -15634.091} C_VEL
LIN {X 0,Y 312.566,Z 345.168,A -85,B 0,C 180,E1 -15637.528,E2 -15637.528} C_VEL
LIN {X 0,Y 312.641,Z 345.159,A -85,B 0,C 180,E1 -15641.657,E2 -15641.657} C_VEL
LIN {X 0,Y 312.697,Z 345.155,A -85,B 0,C 180,E1 -15645.687,E2 -15645.687} C_VEL
LIN {X 0,Y 312.701,Z 345.16,A -85,B 0,C 180,E1 -15649.642,E2 -15649.642} C_VEL
LIN {X 0,Y 312.799,Z 345.137,A -85,B 0,C 180,E1 -15652.253,E2 -15652.253} C_VEL
LIN {X 0,Y 312.694,Z 345.157,A -85,B 0,C 180,E1 -15654.842,E2 -15654.842} C_VEL
LIN {X 0,Y 312.983,Z 345.122,A -85,B 0,C 180,E1 -15658.714,E2 -15658.714} C_VEL
LIN {X 0,Y 312.926,Z 345.123,A -85,B 0,C 180,E1 -15662.575,E2 -15662.575} C_VEL
LIN {X 0,Y 312.845,Z 345.128,A -85,B 0,C 180,E1 -15666.45,E2 -15666.45} C_VEL
LIN {X 0,Y 312.754,Z 345.151,A -85,B 0,C 180,E1 -15669.051,E2 -15669.051} C_VEL
LIN {X 0,Y 312.628,Z 345.163,A -85,B 0,C 180,E1 -15672.992,E2 -15672.992} C_VEL
LIN {X 0,Y 312.571,Z 345.167,A -85,B 0,C 180,E1 -15675.654,E2 -15675.654} C_VEL
LIN {X 0,Y 312.528,Z 345.175,A -85,B 0,C 180,E1 -15679.714,E2 -15679.714} C_VEL
LIN {X 0,Y 312.517,Z 345.181,A -85,B 0,C 180,E1 -15682.775,E2 -15682.775} C_VEL
LIN {X 0,Y 312.485,Z 345.185,A -85,B 0,C 180,E1 -15686.732,E2 -15686.732} C_VEL
LIN {X 0,Y 312.469,Z 345.158,A -85,B 0,C 180,E1 -15689.658,E2 -15689.658} C_VEL
LIN {X 0,Y 312.522,Z 345.182,A -85,B 0,C 180,E1 -15693.689,E2 -15693.689} C_VEL
LIN {X 0,Y 312.516,Z 345.162,A -85,B 0,C 180,E1 -15697.387,E2 -15697.387} C_VEL
LIN {X 0,Y 312.443,Z 345.187,A -85,B 0,C 180,E1 -15700.717,E2 -15700.717} C_VEL
LIN {X 0,Y 312.453,Z 345.191,A -85,B 0,C 180,E1 -15704.21,E2 -15704.21} C_VEL
LIN {X 0,Y 312.457,Z 345.194,A -85,B 0,C 180,E1 -15707.925,E2 -15707.925} C_VEL
LIN {X 0,Y 312.494,Z 345.274,A -85,B 0,C 180,E1 -15710.182,E2 -15710.182} C_VEL
LIN {X 0,Y 313.926,Z 350.283,A -85,B 0,C 180,E1 -15711.928,E2 -15711.928} C_VEL
LIN {X 0,Y 324.086,Z 369.677,A -85,B 0,C 180,E1 -15713.703,E2 -15713.703} C_VEL
LIN {X 0,Y 332.454,Z 388.222,A -85,B 0,C 180,E1 -15715.121,E2 -15715.121} C_VEL
LIN {X 0,Y 333.443,Z 390.587,A -85,B 0,C 180,E1 -15715.287,E2 -15715.287} C_VEL
LIN {X 0,Y 330.592,Z 486.424,A -85,B 0,C 180,E1 -15717.399,E2 -15717.399} C_VEL
LIN {X 0,Y 329.561,Z 501.123,A -85,B 0,C 180,E1 -15717.963,E2 -15717.963} C_VEL
LIN {X 0,Y 328.016,Z 515.706,A -85,B 0,C 180,E1 -15718.786,E2 -15718.786} C_VEL
LIN {X 0,Y 326.614,Z 526.865,A -85,B 0,C 180,E1 -15719.628,E2 -15719.628} C_VEL
LIN {X 0,Y 324.718,Z 539.692,A -85,B 0,C 180,E1 -15720.858,E2 -15720.858} C_VEL
LIN {X 0,Y 322.857,Z 550.169,A -85,B 0,C 180,E1 -15722.094,E2 -15722.094} C_VEL
LIN {X 0,Y 320.794,Z 561.032,A -85,B 0,C 180,E1 -15723.663,E2 -15723.663} C_VEL
LIN {X 0,Y 318.693,Z 571.749,A -85,B 0,C 180,E1 -15725.576,E2 -15725.576} C_VEL
LIN {X 0,Y 316.723,Z 580.56,A -85,B 0,C 180,E1 -15727.494,E2 -15727.494} C_VEL
LIN {X 0,Y 315.026,Z 588.276,A -85,B 0,C 180,E1 -15729.554,E2 -15729.554} C_VEL
LIN {X 0,Y 313.622,Z 594.828,A -85,B 0,C 180,E1 -15731.716,E2 -15731.716} C_VEL
LIN {X 0,Y 312.383,Z 601.051,A -85,B 0,C 180,E1 -15734.337,E2 -15734.337} C_VEL
LIN {X 0,Y 311.462,Z 605.586,A -85,B 0,C 180,E1 -15736.959,E2 -15736.959} C_VEL
LIN {X 0,Y 310.902,Z 608.639,A -85,B 0,C 180,E1 -15739.581,E2 -15739.581} C_VEL
LIN {X 0,Y 310.742,Z 610.313,A -85,B 0,C 180,E1 -15742.201,E2 -15742.201} C_VEL
LIN {X 0,Y 310.727,Z 610.713,A -85,B 0,C 180,E1 -15744.384,E2 -15744.384} C_VEL
LIN {X 0,Y 310.715,Z 610.34,A -85,B 0,C 180,E1 -15746.109,E2 -15746.109} C_VEL
LIN {X 0,Y 310.72,Z 608.717,A -85,B 0,C 180,E1 -15748.704,E2 -15748.704} C_VEL
LIN {X 0,Y 310.957,Z 605.747,A -85,B 0,C 180,E1 -15751.295,E2 -15751.295} C_VEL
LIN {X 0,Y 311.472,Z 601.35,A -85,B 0,C 180,E1 -15753.881,E2 -15753.881} C_VEL
LIN {X 0,Y 312.276,Z 596.979,A -85,B 0,C 180,E1 -15755.813,E2 -15755.813} C_VEL
LIN {X 0,Y 313.166,Z 590.678,A -85,B 0,C 180,E1 -15758.063,E2 -15758.063} C_VEL
LIN {X 0,Y 314.373,Z 582.852,A -85,B 0,C 180,E1 -15760.303,E2 -15760.303} C_VEL
LIN {X 0,Y 315.348,Z 576.152,A -85,B 0,C 180,E1 -15761.897,E2 -15761.897} C_VEL
LIN {X 0,Y 317.152,Z 566.578,A -85,B 0,C 180,E1 -15763.781,E2 -15763.781} C_VEL
LIN {X 0,Y 318.798,Z 555.988,A -85,B 0,C 180,E1 -15765.504,E2 -15765.504} C_VEL
LIN {X 0,Y 320.288,Z 545.553,A -85,B 0,C 180,E1 -15766.902,E2 -15766.902} C_VEL
LIN {X 0,Y 321.985,Z 532.789,A -85,B 0,C 180,E1 -15768.286,E2 -15768.286} C_VEL
LIN {X 0,Y 323.342,Z 520.323,A -85,B 0,C 180,E1 -15769.358,E2 -15769.358} C_VEL
LIN {X 0,Y 324.703,Z 506.405,A -85,B 0,C 180,E1 -15770.262,E2 -15770.262} C_VEL
LIN {X 0,Y 325.594,Z 492.635,A -85,B 0,C 180,E1 -15770.906,E2 -15770.906} C_VEL
LIN {X 0,Y 326.186,Z 478.394,A -85,B 0,C 180,E1 -15771.321,E2 -15771.321} C_VEL
LIN {X 0,Y 328.577,Z 385.589,A -85,B 0,C 180,E1 -15773.332,E2 -15773.332} C_VEL
LIN {X 0,Y 321.145,Z 366.664,A -85,B 0,C 180,E1 -15774.46,E2 -15774.46} C_VEL
LIN {X 0,Y 314.3,Z 351.503,A -85,B 0,C 180,E1 -15775.499,E2 -15775.499} C_VEL
LIN {X 0,Y 313.54,Z 349.582,A -85,B 0,C 180,E1 -15775.641,E2 -15775.641} C_VEL
LIN {X 0,Y 312.564,Z 345.404,A -85,B 0,C 180,E1 -15776.987,E2 -15776.987} C_VEL
LIN {X 0,Y 311.968,Z 345.253,A -85,B 0,C 180,E1 -15777.636,E2 -15777.636} C_VEL
LIN {X 0,Y 308.64,Z 345.658,A -85,B 0,C 180,E1 -15779.714,E2 -15779.714} C_VEL
LIN {X 0,Y 306.408,Z 346.163,A -85,B 0,C 180,E1 -15781.181,E2 -15781.181} C_VEL
LIN {X 0,Y 305.49,Z 346.079,A -85,B 0,C 180,E1 -15782.318,E2 -15782.318} C_VEL
LIN {X 0,Y 305.423,Z 346.063,A -85,B 0,C 180,E1 -15782.702,E2 -15782.702} C_VEL
LIN {X 0,Y 305.464,Z 346.06,A -85,B 0,C 180,E1 -15786.363,E2 -15786.363} C_VEL
LIN {X 0,Y 305.412,Z 346.065,A -85,B 0,C 180,E1 -15790.115,E2 -15790.115} C_VEL
LIN {X 0,Y 305.423,Z 346.064,A -85,B 0,C 180,E1 -15793.656,E2 -15793.656} C_VEL
LIN {X 0,Y 305.437,Z 346.061,A -85,B 0,C 180,E1 -15797.418,E2 -15797.418} C_VEL
LIN {X 0,Y 305.451,Z 346.059,A -85,B 0,C 180,E1 -15801.593,E2 -15801.593} C_VEL
LIN {X 0,Y 305.465,Z 346.061,A -85,B 0,C 180,E1 -15804.886,E2 -15804.886} C_VEL
LIN {X 0,Y 305.444,Z 346.056,A -85,B 0,C 180,E1 -15808.358,E2 -15808.358} C_VEL
LIN {X 0,Y 305.455,Z 346.056,A -85,B 0,C 180,E1 -15811.107,E2 -15811.107} C_VEL
LIN {X 0,Y 305.481,Z 346.053,A -85,B 0,C 180,E1 -15814.079,E2 -15814.079} C_VEL
LIN {X 0,Y 305.476,Z 346.051,A -85,B 0,C 180,E1 -15816.976,E2 -15816.976} C_VEL
LIN {X 0,Y 305.511,Z 346.036,A -85,B 0,C 180,E1 -15821.212,E2 -15821.212} C_VEL
LIN {X 0,Y 305.582,Z 346.042,A -85,B 0,C 180,E1 -15825.345,E2 -15825.345} C_VEL
LIN {X 0,Y 305.627,Z 346.005,A -85,B 0,C 180,E1 -15829.399,E2 -15829.399} C_VEL
LIN {X 0,Y 305.749,Z 346.016,A -85,B 0,C 180,E1 -15832.072,E2 -15832.072} C_VEL
LIN {X 0,Y 305.668,Z 346.032,A -85,B 0,C 180,E1 -15834.723,E2 -15834.723} C_VEL
LIN {X 0,Y 305.941,Z 346,A -85,B 0,C 180,E1 -15838.683,E2 -15838.683} C_VEL
LIN {X 0,Y 305.95,Z 345.99,A -85,B 0,C 180,E1 -15841.316,E2 -15841.316} C_VEL
LIN {X 0,Y 305.79,Z 346.018,A -85,B 0,C 180,E1 -15846.598,E2 -15846.598} C_VEL
LIN {X 0,Y 305.696,Z 346.028,A -85,B 0,C 180,E1 -15849.261,E2 -15849.261} C_VEL
LIN {X 0,Y 305.592,Z 346.043,A -85,B 0,C 180,E1 -15853.296,E2 -15853.296} C_VEL
LIN {X 0,Y 305.596,Z 346.046,A -85,B 0,C 180,E1 -15856.02,E2 -15856.02} C_VEL
LIN {X 0,Y 305.578,Z 346.043,A -85,B 0,C 180,E1 -15859.444,E2 -15859.444} C_VEL
LIN {X 0,Y 305.49,Z 346.054,A -85,B 0,C 180,E1 -15863.04,E2 -15863.04} C_VEL
LIN {X 0,Y 305.502,Z 346.054,A -85,B 0,C 180,E1 -15866.209,E2 -15866.209} C_VEL
LIN {X 0,Y 305.47,Z 346.058,A -85,B 0,C 180,E1 -15869.04,E2 -15869.04} C_VEL
LIN {X 0,Y 305.438,Z 346.063,A -85,B 0,C 180,E1 -15871.952,E2 -15871.952} C_VEL
LIN {X 0,Y 305.464,Z 346.062,A -85,B 0,C 180,E1 -15875.113,E2 -15875.113} C_VEL
LIN {X 0,Y 305.469,Z 346.058,A -85,B 0,C 180,E1 -15878.533,E2 -15878.533} C_VEL
LIN {X 0,Y 305.456,Z 346.063,A -85,B 0,C 180,E1 -15882.586,E2 -15882.586} C_VEL
LIN {X 0,Y 305.426,Z 346.064,A -85,B 0,C 180,E1 -15886.345,E2 -15886.345} C_VEL
LIN {X 0,Y 305.458,Z 346.061,A -85,B 0,C 180,E1 -15889.892,E2 -15889.892} C_VEL
LIN {X 0,Y 305.497,Z 346.083,A -85,B 0,C 180,E1 -15893.506,E2 -15893.506} C_VEL
LIN {X 0,Y 308.102,Z 356.891,A -85,B 0,C 180,E1 -15896.807,E2 -15896.807} C_VEL
LIN {X 0,Y 309.982,Z 364.782,A -85,B 0,C 180,E1 -15899.048,E2 -15899.048} C_VEL
LIN {X 0,Y 316.99,Z 382.039,A -85,B 0,C 180,E1 -15900.172,E2 -15900.172} C_VEL
LIN {X 0,Y 321.684,Z 411.091,A -85,B 0,C 180,E1 -15901.319,E2 -15901.319} C_VEL
LIN {X 0,Y 319.144,Z 503.164,A -85,B 0,C 180,E1 -15903.385,E2 -15903.385} C_VEL
LIN {X 0,Y 318.095,Z 517.702,A -85,B 0,C 180,E1 -15903.952,E2 -15903.952} C_VEL
LIN {X 0,Y 316.683,Z 532.216,A -85,B 0,C 180,E1 -15904.797,E2 -15904.797} C_VEL
LIN {X 0,Y 315.129,Z 545.076,A -85,B 0,C 180,E1 -15905.808,E2 -15905.808} C_VEL
LIN {X 0,Y 313.48,Z 557.651,A -85,B 0,C 180,E1 -15907.079,E2 -15907.079} C_VEL
LIN {X 0,Y 311.687,Z 569.046,A -85,B 0,C 180,E1 -15908.506,E2 -15908.506} C_VEL
LIN {X 0,Y 309.904,Z 579.554,A -85,B 0,C 180,E1 -15910.113,E2 -15910.113} C_VEL
LIN {X 0,Y 308.152,Z 590.008,A -85,B 0,C 180,E1 -15912.068,E2 -15912.068} C_VEL
LIN {X 0,Y 306.741,Z 598.63,A -85,B 0,C 180,E1 -15914.041,E2 -15914.041} C_VEL
LIN {X 0,Y 305.545,Z 606.866,A -85,B 0,C 180,E1 -15916.363,E2 -15916.363} C_VEL
LIN {X 0,Y 304.533,Z 613.489,A -85,B 0,C 180,E1 -15918.687,E2 -15918.687} C_VEL
LIN {X 0,Y 303.95,Z 619.366,A -85,B 0,C 180,E1 -15921.356,E2 -15921.356} C_VEL
LIN {X 0,Y 303.739,Z 622.748,A -85,B 0,C 180,E1 -15923.356,E2 -15923.356} C_VEL
LIN {X 0,Y 303.629,Z 625.908,A -85,B 0,C 180,E1 -15926.018,E2 -15926.018} C_VEL
LIN {X 0,Y 303.576,Z 627.677,A -85,B 0,C 180,E1 -15928.673,E2 -15928.673} C_VEL
LIN {X 0,Y 303.603,Z 628.057,A -85,B 0,C 180,E1 -15930,E2 -15930} C_VEL
LIN {X 0,Y 303.598,Z 627.811,A -85,B 0,C 180,E1 -15932.654,E2 -15932.654} C_VEL
LIN {X 0,Y 303.616,Z 626.23,A -85,B 0,C 180,E1 -15935.313,E2 -15935.313} C_VEL
LIN {X 0,Y 303.912,Z 623.287,A -85,B 0,C 180,E1 -15937.976,E2 -15937.976} C_VEL
LIN {X 0,Y 304.503,Z 618.904,A -85,B 0,C 180,E1 -15940.64,E2 -15940.64} C_VEL
LIN {X 0,Y 305.263,Z 614.582,A -85,B 0,C 180,E1 -15942.634,E2 -15942.634} C_VEL
LIN {X 0,Y 306.516,Z 608.312,A -85,B 0,C 180,E1 -15944.948,E2 -15944.948} C_VEL
LIN {X 0,Y 308.11,Z 600.523,A -85,B 0,C 180,E1 -15947.25,E2 -15947.25} C_VEL
LIN {X 0,Y 309.932,Z 592.409,A -85,B 0,C 180,E1 -15949.196,E2 -15949.196} C_VEL
LIN {X 0,Y 312.075,Z 582.651,A -85,B 0,C 180,E1 -15951.12,E2 -15951.12} C_VEL
LIN {X 0,Y 314.451,Z 571.832,A -85,B 0,C 180,E1 -15952.851,E2 -15952.851} C_VEL
LIN {X 0,Y 316.684,Z 560.253,A -85,B 0,C 180,E1 -15954.362,E2 -15954.362} C_VEL
LIN {X 0,Y 318.687,Z 548.086,A -85,B 0,C 180,E1 -15955.645,E2 -15955.645} C_VEL
LIN {X 0,Y 320.638,Z 535.214,A -85,B 0,C 180,E1 -15956.701,E2 -15956.701} C_VEL
LIN {X 0,Y 322.294,Z 522.033,A -85,B 0,C 180,E1 -15957.518,E2 -15957.518} C_VEL
LIN {X 0,Y 323.625,Z 507.686,A -85,B 0,C 180,E1 -15958.142,E2 -15958.142} C_VEL
LIN {X 0,Y 324.355,Z 491.684,A -85,B 0,C 180,E1 -15958.58,E2 -15958.58} C_VEL
LIN {X 0,Y 326.847,Z 412.79,A -85,B 0,C 180,E1 -15960.31,E2 -15960.31} C_VEL
LIN {X 0,Y 322.813,Z 390.806,A -85,B 0,C 180,E1 -15961.334,E2 -15961.334} C_VEL
LIN {X 0,Y 315.075,Z 373.927,A -85,B 0,C 180,E1 -15962.718,E2 -15962.718} C_VEL
LIN {X 0,Y 310.312,Z 364.07,A -85,B 0,C 180,E1 -15963.613,E2 -15963.613} C_VEL
LIN {X 0,Y 307.323,Z 352.687,A -85,B 0,C 180,E1 -15967.347,E2 -15967.347} C_VEL
LIN {X 0,Y 305.477,Z 346.052,A -85,B 0,C 180,E1 -15969.687,E2 -15969.687} C_VEL
LIN {X 0,Y 305.426,Z 346.061,A -85,B 0,C 180,E1 -15973.655,E2 -15973.655} C_VEL
LIN {X 0,Y 305.456,Z 346.059,A -85,B 0,C 180,E1 -15977.415,E2 -15977.415} C_VEL
LIN {X 0,Y 305.497,Z 346.053,A -85,B 0,C 180,E1 -15981.601,E2 -15981.601} C_VEL
LIN {X 0,Y 305.464,Z 346.061,A -85,B 0,C 180,E1 -15984.887,E2 -15984.887} C_VEL
LIN {X 0,Y 305.443,Z 346.065,A -85,B 0,C 180,E1 -15988.358,E2 -15988.358} C_VEL
LIN {X 0,Y 305.488,Z 346.055,A -85,B 0,C 180,E1 -15991.111,E2 -15991.111} C_VEL
LIN {X 0,Y 305.506,Z 346.047,A -85,B 0,C 180,E1 -15994.082,E2 -15994.082} C_VEL
LIN {X 0,Y 305.484,Z 346.05,A -85,B 0,C 180,E1 -15998.402,E2 -15998.402} C_VEL
LIN {X 0,Y 305.592,Z 346.04,A -85,B 0,C 180,E1 -16001.218,E2 -16001.218} C_VEL
LIN {X 0,Y 305.652,Z 346.036,A -85,B 0,C 180,E1 -16005.349,E2 -16005.349} C_VEL
LIN {X 0,Y 305.638,Z 346.038,A -85,B 0,C 180,E1 -16009.4,E2 -16009.4} C_VEL
LIN {X 0,Y 305.749,Z 346.014,A -85,B 0,C 180,E1 -16012.073,E2 -16012.073} C_VEL
LIN {X 0,Y 305.664,Z 346.033,A -85,B 0,C 180,E1 -16014.723,E2 -16014.723} C_VEL
LIN {X 0,Y 305.95,Z 345.999,A -85,B 0,C 180,E1 -16018.684,E2 -16018.684} C_VEL
LIN {X 0,Y 305.942,Z 345.991,A -85,B 0,C 180,E1 -16021.317,E2 -16021.317} C_VEL
LIN {X 0,Y 305.667,Z 346.034,A -85,B 0,C 180,E1 -16025.277,E2 -16025.277} C_VEL
LIN {X 0,Y 305.75,Z 346.017,A -85,B 0,C 180,E1 -16027.928,E2 -16027.928} C_VEL
LIN {X 0,Y 305.599,Z 346.033,A -85,B 0,C 180,E1 -16031.946,E2 -16031.946} C_VEL
LIN {X 0,Y 305.562,Z 346.047,A -85,B 0,C 180,E1 -16034.979,E2 -16034.979} C_VEL
LIN {X 0,Y 305.502,Z 346.055,A -85,B 0,C 180,E1 -16038.788,E2 -16038.788} C_VEL
LIN {X 0,Y 305.458,Z 346.061,A -85,B 0,C 180,E1 -16043.026,E2 -16043.026} C_VEL
LIN {X 0,Y 305.454,Z 346.061,A -85,B 0,C 180,E1 -16046.19,E2 -16046.19} C_VEL
LIN {X 0,Y 305.426,Z 346.042,A -85,B 0,C 180,E1 -16049.025,E2 -16049.025} C_VEL
LIN {X 0,Y 305.437,Z 346.046,A -85,B 0,C 180,E1 -16051.953,E2 -16051.953} C_VEL
LIN {X 0,Y 305.464,Z 346.047,A -85,B 0,C 180,E1 -16055.114,E2 -16055.114} C_VEL
LIN {X 0,Y 305.436,Z 346.062,A -85,B 0,C 180,E1 -16058.525,E2 -16058.525} C_VEL
LIN {X 0,Y 305.437,Z 346.062,A -85,B 0,C 180,E1 -16062.582,E2 -16062.582} C_VEL
LIN {X 0,Y 305.423,Z 346.055,A -85,B 0,C 180,E1 -16066.344,E2 -16066.344} C_VEL
LIN {X 0,Y 305.418,Z 346.21,A -85,B 0,C 180,E1 -16069.409,E2 -16069.409} C_VEL
LIN {X 0,Y 306.572,Z 350.296,A -85,B 0,C 180,E1 -16070.942,E2 -16070.942} C_VEL
LIN {X 0,Y 316.952,Z 369.631,A -85,B 0,C 180,E1 -16072.839,E2 -16072.839} C_VEL
LIN {X 0,Y 324.77,Z 386.455,A -85,B 0,C 180,E1 -16074.218,E2 -16074.218} C_VEL
LIN {X 0,Y 327.441,Z 392.739,A -85,B 0,C 180,E1 -16074.683,E2 -16074.683} C_VEL
LIN {X 0,Y 324.463,Z 485.803,A -85,B 0,C 180,E1 -16076.751,E2 -16076.751} C_VEL
LIN {X 0,Y 323.543,Z 500.075,A -85,B 0,C 180,E1 -16077.293,E2 -16077.293} C_VEL
LIN {X 0,Y 322.076,Z 513.839,A -85,B 0,C 180,E1 -16078.051,E2 -16078.051} C_VEL
LIN {X 0,Y 320.294,Z 527.273,A -85,B 0,C 180,E1 -16079.06,E2 -16079.06} C_VEL
LIN {X 0,Y 318.452,Z 539.304,A -85,B 0,C 180,E1 -16080.227,E2 -16080.227} C_VEL
LIN {X 0,Y 316.296,Z 551.069,A -85,B 0,C 180,E1 -16081.644,E2 -16081.644} C_VEL
LIN {X 0,Y 314.339,Z 560.831,A -85,B 0,C 180,E1 -16083.079,E2 -16083.079} C_VEL
LIN {X 0,Y 312.137,Z 571.614,A -85,B 0,C 180,E1 -16085.028,E2 -16085.028} C_VEL
LIN {X 0,Y 310.057,Z 580.482,A -85,B 0,C 180,E1 -16086.983,E2 -16086.983} C_VEL
LIN {X 0,Y 308.143,Z 588.798,A -85,B 0,C 180,E1 -16089.248,E2 -16089.248} C_VEL
LIN {X 0,Y 306.792,Z 594.843,A -85,B 0,C 180,E1 -16091.294,E2 -16091.294} C_VEL
LIN {X 0,Y 305.437,Z 601.11,A -85,B 0,C 180,E1 -16093.971,E2 -16093.971} C_VEL
LIN {X 0,Y 304.461,Z 605.697,A -85,B 0,C 180,E1 -16096.654,E2 -16096.654} C_VEL
LIN {X 0,Y 303.841,Z 608.784,A -85,B 0,C 180,E1 -16099.336,E2 -16099.336} C_VEL
LIN {X 0,Y 303.651,Z 610.491,A -85,B 0,C 180,E1 -16102.017,E2 -16102.017} C_VEL
LIN {X 0,Y 303.623,Z 610.897,A -85,B 0,C 180,E1 -16104.464,E2 -16104.464} C_VEL
LIN {X 0,Y 303.628,Z 610.566,A -85,B 0,C 180,E1 -16106.018,E2 -16106.018} C_VEL
LIN {X 0,Y 303.634,Z 608.977,A -85,B 0,C 180,E1 -16108.674,E2 -16108.674} C_VEL
LIN {X 0,Y 303.865,Z 606.04,A -85,B 0,C 180,E1 -16111.325,E2 -16111.325} C_VEL
